emC_LUC[LUC_Num].SCADA.Out.BmsUdcAct	:=	emC_LUC[LUC_Num].BattPLC.CtrlLo.Out.Batt_Sys.BattSysMeasure.UdcAct		;
emC_LUC[LUC_Num].SCADA.Out.BmsIdcAct	:=	emC_LUC[LUC_Num].BattPLC.CtrlLo.Out.Batt_Sys.BattSysMeasure.IdcAct		;
emC_LUC[LUC_Num].SCADA.Out.BmsNomPAct	:=	emC_LUC[LUC_Num].BattPLC.CtrlLo.Out.Batt_Sys.BattSysMeasure.NomPAct		;
emC_LUC[LUC_Num].SCADA.Out.BmsNomEAct	:=	emC_LUC[LUC_Num].BattPLC.CtrlLo.Out.Batt_Sys.BattSysMeasure.NomEAct		;
emC_LUC[LUC_Num].SCADA.Out.BatPNomMaxAct	:=	emC_LUC[LUC_Num].BattPLC.CtrlLo.Out.Batt_Sys.BattSysMeasure.BatPNomMaxAct		;
emC_LUC[LUC_Num].SCADA.Out.BatPNomMinAct	:=	emC_LUC[LUC_Num].BattPLC.CtrlLo.Out.Batt_Sys.BattSysMeasure.BatPNomMinAct		;
emC_LUC[LUC_Num].SCADA.Out.BmsPAct	:=	emC_LUC[LUC_Num].BattPLC.CtrlLo.Out.Batt_Sys.BattSysMeasure.PAct		;
emC_LUC[LUC_Num].SCADA.Out.BmsEAct	:=	emC_LUC[LUC_Num].BattPLC.CtrlLo.Out.Batt_Sys.BattSysMeasure.EAct		;
emC_LUC[LUC_Num].SCADA.Out.BmsSocPctAct	:=	emC_LUC[LUC_Num].BattPLC.CtrlLo.Out.Batt_Sys.BattSysMeasure.SocPctAct		;
emC_LUC[LUC_Num].SCADA.Out.BmsSohAct	:=	emC_LUC[LUC_Num].BattPLC.CtrlLo.Out.Batt_Sys.BattSysMeasure.SohAct		;
emC_LUC[LUC_Num].SCADA.Out.BmsTempMaxAct	:=	emC_LUC[LUC_Num].BattPLC.CtrlLo.Out.Batt_Sys.BattSysMeasure.TempMaxAct		;
emC_LUC[LUC_Num].SCADA.Out.BmsTempMinAct	:=	emC_LUC[LUC_Num].BattPLC.CtrlLo.Out.Batt_Sys.BattSysMeasure.TempMinAct		;
emC_LUC[LUC_Num].SCADA.Out.BmsSyncUSet	:=	emC_LUC[LUC_Num].BattPLC.CtrlLo.Out.Batt_Sys.BattSysMeasure.SyncUSet		;
emC_LUC[LUC_Num].SCADA.Out.BmsHeartBeat	:=	emC_LUC[LUC_Num].BattPLC.CtrlLo.Out.Batt_Sys.BMS_DATA.HeartBeat		;
emC_LUC[LUC_Num].SCADA.Out.BmsVersion	:=	UINT_TO_REAL(emC_LUC[LUC_Num].BattPLC.CtrlLo.Out.Batt_Sys.BMS_DATA.Version	)	;
emC_LUC[LUC_Num].SCADA.Out.BmsRacksNServiceCnt	:=	USINT_TO_REAL(emC_LUC[LUC_Num].BattPLC.CtrlLo.Out.Batt_Sys.BMS_DATA.RacksNServiceCnt)		;
emC_LUC[LUC_Num].SCADA.Out.BmsTotalRackCnt	:=	USINT_TO_REAL(emC_LUC[LUC_Num].BattPLC.CtrlLo.Out.Batt_Sys.BMS_DATA.TotalRackCnt)		;
emC_LUC[LUC_Num].SCADA.Out.BmsPartMinRackCnt	:=	USINT_TO_REAL(emC_LUC[LUC_Num].BattPLC.CtrlLo.Out.Batt_Sys.BMS_DATA.PartMinRackCnt)		;
								
								
								
								
								
emC_LUC[LUC_Num].SCADA.Out.PSStateWord	:=	INT_TO_REAL(emC_LUC[LUC_Num].emPs.PS.PSStateWord)	;
emC_LUC[LUC_Num].SCADA.Out.GCABBStateWord	:=	INT_TO_REAL(emC_LUC[LUC_Num].emPs.PS.ABBStateWord)	;
emC_LUC[LUC_Num].SCADA.Out.GCPAct	:=	emC_LUC[LUC_Num].emPs.PS.GCPAct	;
emC_LUC[LUC_Num].SCADA.Out.GCFAct	:=	emC_LUC[LUC_Num].emPs.PS.GCFAct	;
emC_LUC[LUC_Num].SCADA.Out.GCSNomAct	:=	emC_LUC[LUC_Num].emPs.PS.GCSNomAct	;
emC_LUC[LUC_Num].SCADA.Out.GCQAct	:=	emC_LUC[LUC_Num].emPs.PS.GCQAct	;
emC_LUC[LUC_Num].SCADA.Out.GCPF	:=	emC_LUC[LUC_Num].emPs.PS.GCPF	;
emC_LUC[LUC_Num].SCADA.Out.GCEAct	:=	emC_LUC[LUC_Num].emPs.PS.GCEAct	;
emC_LUC[LUC_Num].SCADA.Out.GCTempAct	:=	emC_LUC[LUC_Num].emPs.PS.TempAct	;
emC_LUC[LUC_Num].SCADA.Out.GCIGBTTempaAct	:=	emC_LUC[LUC_Num].emPs.PS.IGBTTempaAct	;
emC_LUC[LUC_Num].SCADA.Out.GCTrafoTempAct	:=	emC_LUC[LUC_Num].emPs.PS.TrafoTempAct	;
emC_LUC[LUC_Num].SCADA.Out.GCOTTempAct	:=	emC_LUC[LUC_Num].emPs.PS.OTTempAct	;
emC_LUC[LUC_Num].SCADA.Out.GCUAct12	:=	emC_LUC[LUC_Num].emPs.PS.GCUAct12	;
emC_LUC[LUC_Num].SCADA.Out.GCUAct23	:=	emC_LUC[LUC_Num].emPs.PS.GCUAct23	;
emC_LUC[LUC_Num].SCADA.Out.GCUAct13	:=	emC_LUC[LUC_Num].emPs.PS.GCUAct13	;
emC_LUC[LUC_Num].SCADA.Out.GCUAct1N	:=	emC_LUC[LUC_Num].emPs.PS.GCUAct1N	;
emC_LUC[LUC_Num].SCADA.Out.GCUAct2N	:=	emC_LUC[LUC_Num].emPs.PS.GCUAct2N	;
emC_LUC[LUC_Num].SCADA.Out.GCUAct3N	:=	emC_LUC[LUC_Num].emPs.PS.GCUAct3N	;
emC_LUC[LUC_Num].SCADA.Out.GCUAct	:=	emC_LUC[LUC_Num].emPs.PS.GCUAct	;
emC_LUC[LUC_Num].SCADA.Out.GCABBErrorID	:=	emC_LUC[LUC_Num].emPs.PS.GCABBErrorID	;
emC_LUC[LUC_Num].SCADA.Out.GCSysFltCode	:=	UINT_TO_REAL(emC_LUC[LUC_Num].emPs.PS.GCSysFltCode)	;
emC_LUC[LUC_Num].SCADA.Out.I1Act	:=	emC_LUC[LUC_Num].emPs.PS.GCAPhA	;
emC_LUC[LUC_Num].SCADA.Out.I2Act	:=	emC_LUC[LUC_Num].emPs.PS.GCAPhB	;
emC_LUC[LUC_Num].SCADA.Out.I3Act	:=	emC_LUC[LUC_Num].emPs.PS.GCAPhC	;
								
								
								
S_MFI_MNG_16	(MFI_Value:=	emC_LUC[LUC_Num].SCADA.Out.GcSPNomAct	,TimeTag:=Timestamp,IV:=FALSE,CycTrigPa:=FALSE,DeadBTransmitPa:=REAL#0.0,TransmitModePa:= INT#1);	GcSPNomAct_Q	:=	S_MFI_MNG_16.Analog_Output_Q	;
S_MFI_MNG_17	(MFI_Value:=	emC_LUC[LUC_Num].SCADA.Out.GcINomAct	,TimeTag:=Timestamp,IV:=FALSE,CycTrigPa:=FALSE,DeadBTransmitPa:=REAL#0.0,TransmitModePa:= INT#1);	GcINomAct_Q	:=	S_MFI_MNG_17.Analog_Output_Q	;
S_MFI_MNG_18	(MFI_Value:=	emC_LUC[LUC_Num].SCADA.Out.GcUNomAct	,TimeTag:=Timestamp,IV:=FALSE,CycTrigPa:=FALSE,DeadBTransmitPa:=REAL#0.0,TransmitModePa:= INT#1);	GcUNomAct_Q	:=	S_MFI_MNG_18.Analog_Output_Q	;
S_MFI_MNG_19	(MFI_Value:=	emC_LUC[LUC_Num].SCADA.Out.GcFNomAct	,TimeTag:=Timestamp,IV:=FALSE,CycTrigPa:=FALSE,DeadBTransmitPa:=REAL#0.0,TransmitModePa:= INT#1);	GcFNomAct_Q	:=	S_MFI_MNG_19.Analog_Output_Q	;
S_MFI_MNG_20	(MFI_Value:=	emC_LUC[LUC_Num].SCADA.Out.GcModUNomAct	,TimeTag:=Timestamp,IV:=FALSE,CycTrigPa:=FALSE,DeadBTransmitPa:=REAL#0.0,TransmitModePa:= INT#1);	GcModUNomAct_Q	:=	S_MFI_MNG_20.Analog_Output_Q	;
								
S_MFI_MNG_21	(MFI_Value:=	emC_LUC[LUC_Num].SCADA.Out.BmsUdcAct	,TimeTag:=Timestamp,IV:=FALSE,CycTrigPa:=FALSE,DeadBTransmitPa:=REAL#0.0,TransmitModePa:= INT#1);	BmsUdcAct_Q	:=	S_MFI_MNG_21.Analog_Output_Q	;
S_MFI_MNG_22	(MFI_Value:=	emC_LUC[LUC_Num].SCADA.Out.BmsIdcAct	,TimeTag:=Timestamp,IV:=FALSE,CycTrigPa:=FALSE,DeadBTransmitPa:=REAL#0.0,TransmitModePa:= INT#1);	BmsIdcAct_Q	:=	S_MFI_MNG_22.Analog_Output_Q	;
S_MFI_MNG_23	(MFI_Value:=	emC_LUC[LUC_Num].SCADA.Out.BmsNomPAct	,TimeTag:=Timestamp,IV:=FALSE,CycTrigPa:=FALSE,DeadBTransmitPa:=REAL#0.0,TransmitModePa:= INT#1);	BmsNomPAct_Q	:=	S_MFI_MNG_23.Analog_Output_Q	;
S_MFI_MNG_24	(MFI_Value:=	emC_LUC[LUC_Num].SCADA.Out.BmsNomEAct	,TimeTag:=Timestamp,IV:=FALSE,CycTrigPa:=FALSE,DeadBTransmitPa:=REAL#0.0,TransmitModePa:= INT#1);	BmsNomEAct_Q	:=	S_MFI_MNG_24.Analog_Output_Q	;
S_MFI_MNG_25	(MFI_Value:=	emC_LUC[LUC_Num].SCADA.Out.BatPNomMaxAct	,TimeTag:=Timestamp,IV:=FALSE,CycTrigPa:=FALSE,DeadBTransmitPa:=REAL#0.0,TransmitModePa:= INT#1);	BmsBatPNomMaxAct_Q	:=	S_MFI_MNG_25.Analog_Output_Q	;
S_MFI_MNG_26	(MFI_Value:=	emC_LUC[LUC_Num].SCADA.Out.BatPNomMinAct	,TimeTag:=Timestamp,IV:=FALSE,CycTrigPa:=FALSE,DeadBTransmitPa:=REAL#0.0,TransmitModePa:= INT#1);	BmsBatPNomMinAct_Q	:=	S_MFI_MNG_26.Analog_Output_Q	;
S_MFI_MNG_27	(MFI_Value:=	emC_LUC[LUC_Num].SCADA.Out.BmsPAct	,TimeTag:=Timestamp,IV:=FALSE,CycTrigPa:=FALSE,DeadBTransmitPa:=REAL#0.0,TransmitModePa:= INT#1);	BmsPAct_Q	:=	S_MFI_MNG_27.Analog_Output_Q	;
S_MFI_MNG_28	(MFI_Value:=	emC_LUC[LUC_Num].SCADA.Out.BmsEAct	,TimeTag:=Timestamp,IV:=FALSE,CycTrigPa:=FALSE,DeadBTransmitPa:=REAL#0.0,TransmitModePa:= INT#1);	BmsEAct_Q	:=	S_MFI_MNG_28.Analog_Output_Q	;
S_MFI_MNG_29	(MFI_Value:=	emC_LUC[LUC_Num].SCADA.Out.BmsSocPctAct	,TimeTag:=Timestamp,IV:=FALSE,CycTrigPa:=FALSE,DeadBTransmitPa:=REAL#0.0,TransmitModePa:= INT#1);	BatSocAct_Q	:=	S_MFI_MNG_29.Analog_Output_Q	;
S_MFI_MNG_30	(MFI_Value:=	emC_LUC[LUC_Num].SCADA.Out.BmsSohAct	,TimeTag:=Timestamp,IV:=FALSE,CycTrigPa:=FALSE,DeadBTransmitPa:=REAL#0.0,TransmitModePa:= INT#1);	BmsSohAct_Q	:=	S_MFI_MNG_30.Analog_Output_Q	;
S_MFI_MNG_31	(MFI_Value:=	emC_LUC[LUC_Num].SCADA.Out.BmsTempMaxAct	,TimeTag:=Timestamp,IV:=FALSE,CycTrigPa:=FALSE,DeadBTransmitPa:=REAL#0.0,TransmitModePa:= INT#1);	BmsTempMaxAct_Q	:=	S_MFI_MNG_31.Analog_Output_Q	;
S_MFI_MNG_32	(MFI_Value:=	emC_LUC[LUC_Num].SCADA.Out.BmsTempMinAct	,TimeTag:=Timestamp,IV:=FALSE,CycTrigPa:=FALSE,DeadBTransmitPa:=REAL#0.0,TransmitModePa:= INT#1);	BmsTempMinAct_Q	:=	S_MFI_MNG_32.Analog_Output_Q	;
S_MFI_MNG_33	(MFI_Value:=	emC_LUC[LUC_Num].SCADA.Out.BmsSyncUSet	,TimeTag:=Timestamp,IV:=FALSE,CycTrigPa:=FALSE,DeadBTransmitPa:=REAL#0.0,TransmitModePa:= INT#1);	BmsSyncUSet_Q	:=	S_MFI_MNG_33.Analog_Output_Q	;
S_MFI_MNG_34	(MFI_Value:=	emC_LUC[LUC_Num].SCADA.Out.BmsHeartBeat	,TimeTag:=Timestamp,IV:=FALSE,CycTrigPa:=FALSE,DeadBTransmitPa:=REAL#0.0,TransmitModePa:= INT#1);	BmsHeartBeat_Q	:=	S_MFI_MNG_34.Analog_Output_Q	;							
S_MFI_MNG_37	(MFI_Value:=	emC_LUC[LUC_Num].SCADA.Out.BmsVersion	,TimeTag:=Timestamp,IV:=FALSE,CycTrigPa:=FALSE,DeadBTransmitPa:=REAL#0.0,TransmitModePa:= INT#1);	BmsVersion_Q	:=	S_MFI_MNG_37.Analog_Output_Q	;
S_MFI_MNG_38	(MFI_Value:=	emC_LUC[LUC_Num].SCADA.Out.BmsRacksNServiceCnt	,TimeTag:=Timestamp,IV:=FALSE,CycTrigPa:=FALSE,DeadBTransmitPa:=REAL#0.0,TransmitModePa:= INT#1);	BmsRacksNServiceCnt_Q	:=	S_MFI_MNG_38.Analog_Output_Q	;
S_MFI_MNG_39	(MFI_Value:=	emC_LUC[LUC_Num].SCADA.Out.BmsTotalRackCnt	,TimeTag:=Timestamp,IV:=FALSE,CycTrigPa:=FALSE,DeadBTransmitPa:=REAL#0.0,TransmitModePa:= INT#1);	BmsTotalRackCnt_Q	:=	S_MFI_MNG_39.Analog_Output_Q	;
S_MFI_MNG_40	(MFI_Value:=	emC_LUC[LUC_Num].SCADA.Out.BmsPartMinRackCnt	,TimeTag:=Timestamp,IV:=FALSE,CycTrigPa:=FALSE,DeadBTransmitPa:=REAL#0.0,TransmitModePa:= INT#1);	BmsPartMinRackCnt_Q	:=	S_MFI_MNG_40.Analog_Output_Q	;
								
								
								
							
S_MFI_MNG_41	(MFI_Value:=	emC_LUC[LUC_Num].SCADA.Out.PSStateWord	,TimeTag:=Timestamp,IV:=FALSE,CycTrigPa:=FALSE,DeadBTransmitPa:=REAL#0.0,TransmitModePa:= INT#1);	PSStateWord_Q	:=	S_MFI_MNG_41.Analog_Output_Q	;
S_MFI_MNG_42	(MFI_Value:=	emC_LUC[LUC_Num].SCADA.Out.GCABBStateWord	,TimeTag:=Timestamp,IV:=FALSE,CycTrigPa:=FALSE,DeadBTransmitPa:=REAL#0.0,TransmitModePa:= INT#1);	ABBStateWord_Q	:=	S_MFI_MNG_42.Analog_Output_Q	;
S_MFI_MNG_43	(MFI_Value:=	emC_LUC[LUC_Num].SCADA.Out.GCPAct	,TimeTag:=Timestamp,IV:=FALSE,CycTrigPa:=FALSE,DeadBTransmitPa:=REAL#0.0,TransmitModePa:= INT#1);	GCPAct_Q	:=	S_MFI_MNG_43.Analog_Output_Q	;
S_MFI_MNG_44	(MFI_Value:=	emC_LUC[LUC_Num].SCADA.Out.GCFAct	,TimeTag:=Timestamp,IV:=FALSE,CycTrigPa:=FALSE,DeadBTransmitPa:=REAL#0.0,TransmitModePa:= INT#1);	GCFAct_Q	:=	S_MFI_MNG_44.Analog_Output_Q	;
S_MFI_MNG_45	(MFI_Value:=	emC_LUC[LUC_Num].SCADA.Out.GCSNomAct	,TimeTag:=Timestamp,IV:=FALSE,CycTrigPa:=FALSE,DeadBTransmitPa:=REAL#0.0,TransmitModePa:= INT#1);	GCSNomAct_Q	:=	S_MFI_MNG_45.Analog_Output_Q	;
S_MFI_MNG_46	(MFI_Value:=	emC_LUC[LUC_Num].SCADA.Out.GCQAct	,TimeTag:=Timestamp,IV:=FALSE,CycTrigPa:=FALSE,DeadBTransmitPa:=REAL#0.0,TransmitModePa:= INT#1);	GCQAct_Q	:=	S_MFI_MNG_46.Analog_Output_Q	;
S_MFI_MNG_47	(MFI_Value:=	emC_LUC[LUC_Num].SCADA.Out.GCPF	,TimeTag:=Timestamp,IV:=FALSE,CycTrigPa:=FALSE,DeadBTransmitPa:=REAL#0.0,TransmitModePa:= INT#1);	GCPF_Q	:=	S_MFI_MNG_47.Analog_Output_Q	;
S_MFI_MNG_48	(MFI_Value:=	emC_LUC[LUC_Num].SCADA.Out.GCEAct	,TimeTag:=Timestamp,IV:=FALSE,CycTrigPa:=FALSE,DeadBTransmitPa:=REAL#0.0,TransmitModePa:= INT#1);	GCEAct_Q	:=	S_MFI_MNG_48.Analog_Output_Q	;
S_MFI_MNG_49	(MFI_Value:=	emC_LUC[LUC_Num].SCADA.Out.GCTempAct	,TimeTag:=Timestamp,IV:=FALSE,CycTrigPa:=FALSE,DeadBTransmitPa:=REAL#0.0,TransmitModePa:= INT#1);	TempAct_Q	:=	S_MFI_MNG_49.Analog_Output_Q	;
S_MFI_MNG_50	(MFI_Value:=	emC_LUC[LUC_Num].SCADA.Out.GCIGBTTempaAct	,TimeTag:=Timestamp,IV:=FALSE,CycTrigPa:=FALSE,DeadBTransmitPa:=REAL#0.0,TransmitModePa:= INT#1);	IGBTTempaAct_Q	:=	S_MFI_MNG_50.Analog_Output_Q	;
S_MFI_MNG_51	(MFI_Value:=	emC_LUC[LUC_Num].SCADA.Out.GCTrafoTempAct	,TimeTag:=Timestamp,IV:=FALSE,CycTrigPa:=FALSE,DeadBTransmitPa:=REAL#0.0,TransmitModePa:= INT#1);	TrafoTempAct_Q	:=	S_MFI_MNG_51.Analog_Output_Q	;
S_MFI_MNG_52	(MFI_Value:=	emC_LUC[LUC_Num].SCADA.Out.GCOTTempAct	,TimeTag:=Timestamp,IV:=FALSE,CycTrigPa:=FALSE,DeadBTransmitPa:=REAL#0.0,TransmitModePa:= INT#1);	OTTempAct_Q	:=	S_MFI_MNG_52.Analog_Output_Q	;
S_MFI_MNG_53	(MFI_Value:=	emC_LUC[LUC_Num].SCADA.Out.GCUAct12	,TimeTag:=Timestamp,IV:=FALSE,CycTrigPa:=FALSE,DeadBTransmitPa:=REAL#0.0,TransmitModePa:= INT#1);	GCUAct12_Q	:=	S_MFI_MNG_53.Analog_Output_Q	;
S_MFI_MNG_54	(MFI_Value:=	emC_LUC[LUC_Num].SCADA.Out.GCUAct23	,TimeTag:=Timestamp,IV:=FALSE,CycTrigPa:=FALSE,DeadBTransmitPa:=REAL#0.0,TransmitModePa:= INT#1);	GCUAct23_Q	:=	S_MFI_MNG_54.Analog_Output_Q	;
S_MFI_MNG_55	(MFI_Value:=	emC_LUC[LUC_Num].SCADA.Out.GCUAct13	,TimeTag:=Timestamp,IV:=FALSE,CycTrigPa:=FALSE,DeadBTransmitPa:=REAL#0.0,TransmitModePa:= INT#1);	GCUAct13_Q	:=	S_MFI_MNG_55.Analog_Output_Q	;
S_MFI_MNG_56	(MFI_Value:=	emC_LUC[LUC_Num].SCADA.Out.GCUAct1N	,TimeTag:=Timestamp,IV:=FALSE,CycTrigPa:=FALSE,DeadBTransmitPa:=REAL#0.0,TransmitModePa:= INT#1);	GCUAct1N_Q	:=	S_MFI_MNG_56.Analog_Output_Q	;
S_MFI_MNG_57	(MFI_Value:=	emC_LUC[LUC_Num].SCADA.Out.GCUAct2N	,TimeTag:=Timestamp,IV:=FALSE,CycTrigPa:=FALSE,DeadBTransmitPa:=REAL#0.0,TransmitModePa:= INT#1);	GCUAct2N_Q	:=	S_MFI_MNG_57.Analog_Output_Q	;
S_MFI_MNG_58	(MFI_Value:=	emC_LUC[LUC_Num].SCADA.Out.GCUAct3N	,TimeTag:=Timestamp,IV:=FALSE,CycTrigPa:=FALSE,DeadBTransmitPa:=REAL#0.0,TransmitModePa:= INT#1);	GCUAct3N_Q	:=	S_MFI_MNG_58.Analog_Output_Q	;
S_MFI_MNG_59	(MFI_Value:=	emC_LUC[LUC_Num].SCADA.Out.GCUAct	,TimeTag:=Timestamp,IV:=FALSE,CycTrigPa:=FALSE,DeadBTransmitPa:=REAL#0.0,TransmitModePa:= INT#1);	GCUAct_Q	:=	S_MFI_MNG_59.Analog_Output_Q	;
S_MFI_MNG_60	(MFI_Value:=	emC_LUC[LUC_Num].SCADA.Out.GCABBErrorID	,TimeTag:=Timestamp,IV:=FALSE,CycTrigPa:=FALSE,DeadBTransmitPa:=REAL#0.0,TransmitModePa:= INT#1);	GCABBErrorID_Q	:=	S_MFI_MNG_60.Analog_Output_Q	;
S_MFI_MNG_61	(MFI_Value:=	emC_LUC[LUC_Num].SCADA.Out.GCSysFltCode	,TimeTag:=Timestamp,IV:=FALSE,CycTrigPa:=FALSE,DeadBTransmitPa:=REAL#0.0,TransmitModePa:= INT#1);	GCSysFltCode_Q	:=	S_MFI_MNG_61.Analog_Output_Q	;
								
S_MFI_MNG_62	(MFI_Value:=	emC_LUC[LUC_Num].SCADA.Out.I1Act	,TimeTag:=Timestamp,IV:=FALSE,CycTrigPa:=FALSE,DeadBTransmitPa:=REAL#0.0,TransmitModePa:= INT#1);	GCI1_Q	:=	S_MFI_MNG_62.Analog_Output_Q	;
S_MFI_MNG_63	(MFI_Value:=	emC_LUC[LUC_Num].SCADA.Out.I2Act	,TimeTag:=Timestamp,IV:=FALSE,CycTrigPa:=FALSE,DeadBTransmitPa:=REAL#0.0,TransmitModePa:= INT#1);	GCI2_Q	:=	S_MFI_MNG_63.Analog_Output_Q	;
S_MFI_MNG_64	(MFI_Value:=	emC_LUC[LUC_Num].SCADA.Out.I3Act	,TimeTag:=Timestamp,IV:=FALSE,CycTrigPa:=FALSE,DeadBTransmitPa:=REAL#0.0,TransmitModePa:= INT#1);	GCI3_Q	:=	S_MFI_MNG_64.Analog_Output_Q	;
S_MFI_MNG_65	(MFI_Value:=	emC_LUC[LUC_Num].SCADA.Out.IAvgAct	,TimeTag:=Timestamp,IV:=FALSE,CycTrigPa:=FALSE,DeadBTransmitPa:=REAL#0.0,TransmitModePa:= INT#1);	GCIAvgAct_Q	:=	S_MFI_MNG_64.Analog_Output_Q	;
								
								
								
								
S_SPI_MNG_301	(Digital_Feedback_Value:=	emC_LUC[LUC_Num].SCADA.Out.Rk[1].OnlineSt	,TimeTag:=Timestamp,IV:=FALSE);	Rk1OnlineSt_Q	:=	S_SPI_MNG_301.Digital_Feedback_Q	;
S_SPI_MNG_302	(Digital_Feedback_Value:=	emC_LUC[LUC_Num].SCADA.Out.Rk[1].FaultSt	,TimeTag:=Timestamp,IV:=FALSE);	Rk1FaultSt_Q	:=	S_SPI_MNG_302.Digital_Feedback_Q	;
S_MFI_MNG_303	(MFI_Value:=	emC_LUC[LUC_Num].SCADA.Out.Rk[1].SoCAct	,TimeTag:=Timestamp,IV:=FALSE,CycTrigPa:=FALSE,DeadBTransmitPa:=REAL#0.0,TransmitModePa:= INT#1);	Rk1SoCAct_Q	:=	S_MFI_MNG_303.Analog_Output_Q	;
S_MFI_MNG_304	(MFI_Value:=	emC_LUC[LUC_Num].SCADA.Out.Rk[1].SoHAct	,TimeTag:=Timestamp,IV:=FALSE,CycTrigPa:=FALSE,DeadBTransmitPa:=REAL#0.0,TransmitModePa:= INT#1);	Rk1SoHAct_Q	:=	S_MFI_MNG_304.Analog_Output_Q	;
S_MFI_MNG_305	(MFI_Value:=	emC_LUC[LUC_Num].SCADA.Out.Rk[1].UAct	,TimeTag:=Timestamp,IV:=FALSE,CycTrigPa:=FALSE,DeadBTransmitPa:=REAL#0.0,TransmitModePa:= INT#1);	Rk1UAct_Q	:=	S_MFI_MNG_305.Analog_Output_Q	;
S_MFI_MNG_306	(MFI_Value:=	emC_LUC[LUC_Num].SCADA.Out.Rk[1].IAct	,TimeTag:=Timestamp,IV:=FALSE,CycTrigPa:=FALSE,DeadBTransmitPa:=REAL#0.0,TransmitModePa:= INT#1);	Rk1IAct_Q	:=	S_MFI_MNG_306.Analog_Output_Q	;
S_MFI_MNG_307	(MFI_Value:=	emC_LUC[LUC_Num].SCADA.Out.Rk[1].TempAct	,TimeTag:=Timestamp,IV:=FALSE,CycTrigPa:=FALSE,DeadBTransmitPa:=REAL#0.0,TransmitModePa:= INT#1);	Rk1TempAct_Q	:=	S_MFI_MNG_307.Analog_Output_Q	;
S_SPI_MNG_308	(Digital_Feedback_Value:=	emC_LUC[LUC_Num].SCADA.Out.Rk[2].OnlineSt	,TimeTag:=Timestamp,IV:=FALSE);	Rk2OnlineSt_Q	:=	S_SPI_MNG_308.Digital_Feedback_Q	;
S_SPI_MNG_309	(Digital_Feedback_Value:=	emC_LUC[LUC_Num].SCADA.Out.Rk[2].FaultSt	,TimeTag:=Timestamp,IV:=FALSE);	Rk2FaultSt_Q	:=	S_SPI_MNG_309.Digital_Feedback_Q	;
S_MFI_MNG_310	(MFI_Value:=	emC_LUC[LUC_Num].SCADA.Out.Rk[2].SoCAct	,TimeTag:=Timestamp,IV:=FALSE,CycTrigPa:=FALSE,DeadBTransmitPa:=REAL#0.0,TransmitModePa:= INT#1);	Rk2SoCAct_Q	:=	S_MFI_MNG_310.Analog_Output_Q	;
S_MFI_MNG_311	(MFI_Value:=	emC_LUC[LUC_Num].SCADA.Out.Rk[2].SoHAct	,TimeTag:=Timestamp,IV:=FALSE,CycTrigPa:=FALSE,DeadBTransmitPa:=REAL#0.0,TransmitModePa:= INT#1);	Rk2SoHAct_Q	:=	S_MFI_MNG_311.Analog_Output_Q	;
S_MFI_MNG_312	(MFI_Value:=	emC_LUC[LUC_Num].SCADA.Out.Rk[2].UAct	,TimeTag:=Timestamp,IV:=FALSE,CycTrigPa:=FALSE,DeadBTransmitPa:=REAL#0.0,TransmitModePa:= INT#1);	Rk2UAct_Q	:=	S_MFI_MNG_312.Analog_Output_Q	;
S_MFI_MNG_313	(MFI_Value:=	emC_LUC[LUC_Num].SCADA.Out.Rk[2].IAct	,TimeTag:=Timestamp,IV:=FALSE,CycTrigPa:=FALSE,DeadBTransmitPa:=REAL#0.0,TransmitModePa:= INT#1);	Rk2IAct_Q	:=	S_MFI_MNG_313.Analog_Output_Q	;
S_MFI_MNG_314	(MFI_Value:=	emC_LUC[LUC_Num].SCADA.Out.Rk[2].TempAct	,TimeTag:=Timestamp,IV:=FALSE,CycTrigPa:=FALSE,DeadBTransmitPa:=REAL#0.0,TransmitModePa:= INT#1);	Rk2TempAct_Q	:=	S_MFI_MNG_314.Analog_Output_Q	;
S_SPI_MNG_315	(Digital_Feedback_Value:=	emC_LUC[LUC_Num].SCADA.Out.Rk[3].OnlineSt	,TimeTag:=Timestamp,IV:=FALSE);	Rk3OnlineSt_Q	:=	S_SPI_MNG_315.Digital_Feedback_Q	;
S_SPI_MNG_316	(Digital_Feedback_Value:=	emC_LUC[LUC_Num].SCADA.Out.Rk[3].FaultSt	,TimeTag:=Timestamp,IV:=FALSE);	Rk3FaultSt_Q	:=	S_SPI_MNG_316.Digital_Feedback_Q	;
S_MFI_MNG_317	(MFI_Value:=	emC_LUC[LUC_Num].SCADA.Out.Rk[3].SoCAct	,TimeTag:=Timestamp,IV:=FALSE,CycTrigPa:=FALSE,DeadBTransmitPa:=REAL#0.0,TransmitModePa:= INT#1);	Rk3SoCAct_Q	:=	S_MFI_MNG_317.Analog_Output_Q	;
S_MFI_MNG_318	(MFI_Value:=	emC_LUC[LUC_Num].SCADA.Out.Rk[3].SoHAct	,TimeTag:=Timestamp,IV:=FALSE,CycTrigPa:=FALSE,DeadBTransmitPa:=REAL#0.0,TransmitModePa:= INT#1);	Rk3SoHAct_Q	:=	S_MFI_MNG_318.Analog_Output_Q	;
S_MFI_MNG_319	(MFI_Value:=	emC_LUC[LUC_Num].SCADA.Out.Rk[3].UAct	,TimeTag:=Timestamp,IV:=FALSE,CycTrigPa:=FALSE,DeadBTransmitPa:=REAL#0.0,TransmitModePa:= INT#1);	Rk3UAct_Q	:=	S_MFI_MNG_319.Analog_Output_Q	;
S_MFI_MNG_320	(MFI_Value:=	emC_LUC[LUC_Num].SCADA.Out.Rk[3].IAct	,TimeTag:=Timestamp,IV:=FALSE,CycTrigPa:=FALSE,DeadBTransmitPa:=REAL#0.0,TransmitModePa:= INT#1);	Rk3IAct_Q	:=	S_MFI_MNG_320.Analog_Output_Q	;
S_MFI_MNG_321	(MFI_Value:=	emC_LUC[LUC_Num].SCADA.Out.Rk[3].TempAct	,TimeTag:=Timestamp,IV:=FALSE,CycTrigPa:=FALSE,DeadBTransmitPa:=REAL#0.0,TransmitModePa:= INT#1);	Rk3TempAct_Q	:=	S_MFI_MNG_321.Analog_Output_Q	;
S_SPI_MNG_322	(Digital_Feedback_Value:=	emC_LUC[LUC_Num].SCADA.Out.Rk[4].OnlineSt	,TimeTag:=Timestamp,IV:=FALSE);	Rk4OnlineSt_Q	:=	S_SPI_MNG_322.Digital_Feedback_Q	;
S_SPI_MNG_323	(Digital_Feedback_Value:=	emC_LUC[LUC_Num].SCADA.Out.Rk[4].FaultSt	,TimeTag:=Timestamp,IV:=FALSE);	Rk4FaultSt_Q	:=	S_SPI_MNG_323.Digital_Feedback_Q	;
S_MFI_MNG_324	(MFI_Value:=	emC_LUC[LUC_Num].SCADA.Out.Rk[4].SoCAct	,TimeTag:=Timestamp,IV:=FALSE,CycTrigPa:=FALSE,DeadBTransmitPa:=REAL#0.0,TransmitModePa:= INT#1);	Rk4SoCAct_Q	:=	S_MFI_MNG_324.Analog_Output_Q	;
S_MFI_MNG_325	(MFI_Value:=	emC_LUC[LUC_Num].SCADA.Out.Rk[4].SoHAct	,TimeTag:=Timestamp,IV:=FALSE,CycTrigPa:=FALSE,DeadBTransmitPa:=REAL#0.0,TransmitModePa:= INT#1);	Rk4SoHAct_Q	:=	S_MFI_MNG_325.Analog_Output_Q	;
S_MFI_MNG_326	(MFI_Value:=	emC_LUC[LUC_Num].SCADA.Out.Rk[4].UAct	,TimeTag:=Timestamp,IV:=FALSE,CycTrigPa:=FALSE,DeadBTransmitPa:=REAL#0.0,TransmitModePa:= INT#1);	Rk4UAct_Q	:=	S_MFI_MNG_326.Analog_Output_Q	;
S_MFI_MNG_327	(MFI_Value:=	emC_LUC[LUC_Num].SCADA.Out.Rk[4].IAct	,TimeTag:=Timestamp,IV:=FALSE,CycTrigPa:=FALSE,DeadBTransmitPa:=REAL#0.0,TransmitModePa:= INT#1);	Rk4IAct_Q	:=	S_MFI_MNG_327.Analog_Output_Q	;
S_MFI_MNG_328	(MFI_Value:=	emC_LUC[LUC_Num].SCADA.Out.Rk[4].TempAct	,TimeTag:=Timestamp,IV:=FALSE,CycTrigPa:=FALSE,DeadBTransmitPa:=REAL#0.0,TransmitModePa:= INT#1);	Rk4TempAct_Q	:=	S_MFI_MNG_328.Analog_Output_Q	;
S_SPI_MNG_329	(Digital_Feedback_Value:=	emC_LUC[LUC_Num].SCADA.Out.Rk[5].OnlineSt	,TimeTag:=Timestamp,IV:=FALSE);	Rk5OnlineSt_Q	:=	S_SPI_MNG_329.Digital_Feedback_Q	;
S_SPI_MNG_330	(Digital_Feedback_Value:=	emC_LUC[LUC_Num].SCADA.Out.Rk[5].FaultSt	,TimeTag:=Timestamp,IV:=FALSE);	Rk5FaultSt_Q	:=	S_SPI_MNG_330.Digital_Feedback_Q	;
S_MFI_MNG_331	(MFI_Value:=	emC_LUC[LUC_Num].SCADA.Out.Rk[5].SoCAct	,TimeTag:=Timestamp,IV:=FALSE,CycTrigPa:=FALSE,DeadBTransmitPa:=REAL#0.0,TransmitModePa:= INT#1);	Rk5SoCAct_Q	:=	S_MFI_MNG_331.Analog_Output_Q	;
S_MFI_MNG_332	(MFI_Value:=	emC_LUC[LUC_Num].SCADA.Out.Rk[5].SoHAct	,TimeTag:=Timestamp,IV:=FALSE,CycTrigPa:=FALSE,DeadBTransmitPa:=REAL#0.0,TransmitModePa:= INT#1);	Rk5SoHAct_Q	:=	S_MFI_MNG_332.Analog_Output_Q	;
S_MFI_MNG_333	(MFI_Value:=	emC_LUC[LUC_Num].SCADA.Out.Rk[5].UAct	,TimeTag:=Timestamp,IV:=FALSE,CycTrigPa:=FALSE,DeadBTransmitPa:=REAL#0.0,TransmitModePa:= INT#1);	Rk5UAct_Q	:=	S_MFI_MNG_333.Analog_Output_Q	;
S_MFI_MNG_334	(MFI_Value:=	emC_LUC[LUC_Num].SCADA.Out.Rk[5].IAct	,TimeTag:=Timestamp,IV:=FALSE,CycTrigPa:=FALSE,DeadBTransmitPa:=REAL#0.0,TransmitModePa:= INT#1);	Rk5IAct_Q	:=	S_MFI_MNG_334.Analog_Output_Q	;
S_MFI_MNG_335	(MFI_Value:=	emC_LUC[LUC_Num].SCADA.Out.Rk[5].TempAct	,TimeTag:=Timestamp,IV:=FALSE,CycTrigPa:=FALSE,DeadBTransmitPa:=REAL#0.0,TransmitModePa:= INT#1);	Rk5TempAct_Q	:=	S_MFI_MNG_335.Analog_Output_Q	;
S_SPI_MNG_336	(Digital_Feedback_Value:=	emC_LUC[LUC_Num].SCADA.Out.Rk[6].OnlineSt	,TimeTag:=Timestamp,IV:=FALSE);	Rk6OnlineSt_Q	:=	S_SPI_MNG_336.Digital_Feedback_Q	;
S_SPI_MNG_337	(Digital_Feedback_Value:=	emC_LUC[LUC_Num].SCADA.Out.Rk[6].FaultSt	,TimeTag:=Timestamp,IV:=FALSE);	Rk6FaultSt_Q	:=	S_SPI_MNG_337.Digital_Feedback_Q	;
S_MFI_MNG_338	(MFI_Value:=	emC_LUC[LUC_Num].SCADA.Out.Rk[6].SoCAct	,TimeTag:=Timestamp,IV:=FALSE,CycTrigPa:=FALSE,DeadBTransmitPa:=REAL#0.0,TransmitModePa:= INT#1);	Rk6SoCAct_Q	:=	S_MFI_MNG_338.Analog_Output_Q	;
S_MFI_MNG_339	(MFI_Value:=	emC_LUC[LUC_Num].SCADA.Out.Rk[6].SoHAct	,TimeTag:=Timestamp,IV:=FALSE,CycTrigPa:=FALSE,DeadBTransmitPa:=REAL#0.0,TransmitModePa:= INT#1);	Rk6SoHAct_Q	:=	S_MFI_MNG_339.Analog_Output_Q	;
S_MFI_MNG_340	(MFI_Value:=	emC_LUC[LUC_Num].SCADA.Out.Rk[6].UAct	,TimeTag:=Timestamp,IV:=FALSE,CycTrigPa:=FALSE,DeadBTransmitPa:=REAL#0.0,TransmitModePa:= INT#1);	Rk6UAct_Q	:=	S_MFI_MNG_340.Analog_Output_Q	;
S_MFI_MNG_341	(MFI_Value:=	emC_LUC[LUC_Num].SCADA.Out.Rk[6].IAct	,TimeTag:=Timestamp,IV:=FALSE,CycTrigPa:=FALSE,DeadBTransmitPa:=REAL#0.0,TransmitModePa:= INT#1);	Rk6IAct_Q	:=	S_MFI_MNG_341.Analog_Output_Q	;
S_MFI_MNG_342	(MFI_Value:=	emC_LUC[LUC_Num].SCADA.Out.Rk[6].TempAct	,TimeTag:=Timestamp,IV:=FALSE,CycTrigPa:=FALSE,DeadBTransmitPa:=REAL#0.0,TransmitModePa:= INT#1);	Rk6TempAct_Q	:=	S_MFI_MNG_342.Analog_Output_Q	;
S_SPI_MNG_343	(Digital_Feedback_Value:=	emC_LUC[LUC_Num].SCADA.Out.Rk[7].OnlineSt	,TimeTag:=Timestamp,IV:=FALSE);	Rk7OnlineSt_Q	:=	S_SPI_MNG_343.Digital_Feedback_Q	;
S_SPI_MNG_344	(Digital_Feedback_Value:=	emC_LUC[LUC_Num].SCADA.Out.Rk[7].FaultSt	,TimeTag:=Timestamp,IV:=FALSE);	Rk7FaultSt_Q	:=	S_SPI_MNG_344.Digital_Feedback_Q	;
S_MFI_MNG_345	(MFI_Value:=	emC_LUC[LUC_Num].SCADA.Out.Rk[7].SoCAct	,TimeTag:=Timestamp,IV:=FALSE,CycTrigPa:=FALSE,DeadBTransmitPa:=REAL#0.0,TransmitModePa:= INT#1);	Rk7SoCAct_Q	:=	S_MFI_MNG_345.Analog_Output_Q	;
S_MFI_MNG_346	(MFI_Value:=	emC_LUC[LUC_Num].SCADA.Out.Rk[7].SoHAct	,TimeTag:=Timestamp,IV:=FALSE,CycTrigPa:=FALSE,DeadBTransmitPa:=REAL#0.0,TransmitModePa:= INT#1);	Rk7SoHAct_Q	:=	S_MFI_MNG_346.Analog_Output_Q	;
S_MFI_MNG_347	(MFI_Value:=	emC_LUC[LUC_Num].SCADA.Out.Rk[7].UAct	,TimeTag:=Timestamp,IV:=FALSE,CycTrigPa:=FALSE,DeadBTransmitPa:=REAL#0.0,TransmitModePa:= INT#1);	Rk7UAct_Q	:=	S_MFI_MNG_347.Analog_Output_Q	;
S_MFI_MNG_348	(MFI_Value:=	emC_LUC[LUC_Num].SCADA.Out.Rk[7].IAct	,TimeTag:=Timestamp,IV:=FALSE,CycTrigPa:=FALSE,DeadBTransmitPa:=REAL#0.0,TransmitModePa:= INT#1);	Rk7IAct_Q	:=	S_MFI_MNG_348.Analog_Output_Q	;
S_MFI_MNG_349	(MFI_Value:=	emC_LUC[LUC_Num].SCADA.Out.Rk[7].TempAct	,TimeTag:=Timestamp,IV:=FALSE,CycTrigPa:=FALSE,DeadBTransmitPa:=REAL#0.0,TransmitModePa:= INT#1);	Rk7TempAct_Q	:=	S_MFI_MNG_349.Analog_Output_Q	;
S_SPI_MNG_350	(Digital_Feedback_Value:=	emC_LUC[LUC_Num].SCADA.Out.Rk[8].OnlineSt	,TimeTag:=Timestamp,IV:=FALSE);	Rk8OnlineSt_Q	:=	S_SPI_MNG_350.Digital_Feedback_Q	;
S_SPI_MNG_351	(Digital_Feedback_Value:=	emC_LUC[LUC_Num].SCADA.Out.Rk[8].FaultSt	,TimeTag:=Timestamp,IV:=FALSE);	Rk8FaultSt_Q	:=	S_SPI_MNG_351.Digital_Feedback_Q	;
S_MFI_MNG_352	(MFI_Value:=	emC_LUC[LUC_Num].SCADA.Out.Rk[8].SoCAct	,TimeTag:=Timestamp,IV:=FALSE,CycTrigPa:=FALSE,DeadBTransmitPa:=REAL#0.0,TransmitModePa:= INT#1);	Rk8SoCAct_Q	:=	S_MFI_MNG_352.Analog_Output_Q	;
S_MFI_MNG_353	(MFI_Value:=	emC_LUC[LUC_Num].SCADA.Out.Rk[8].SoHAct	,TimeTag:=Timestamp,IV:=FALSE,CycTrigPa:=FALSE,DeadBTransmitPa:=REAL#0.0,TransmitModePa:= INT#1);	Rk8SoHAct_Q	:=	S_MFI_MNG_353.Analog_Output_Q	;
S_MFI_MNG_354	(MFI_Value:=	emC_LUC[LUC_Num].SCADA.Out.Rk[8].UAct	,TimeTag:=Timestamp,IV:=FALSE,CycTrigPa:=FALSE,DeadBTransmitPa:=REAL#0.0,TransmitModePa:= INT#1);	Rk8UAct_Q	:=	S_MFI_MNG_354.Analog_Output_Q	;
S_MFI_MNG_355	(MFI_Value:=	emC_LUC[LUC_Num].SCADA.Out.Rk[8].IAct	,TimeTag:=Timestamp,IV:=FALSE,CycTrigPa:=FALSE,DeadBTransmitPa:=REAL#0.0,TransmitModePa:= INT#1);	Rk8IAct_Q	:=	S_MFI_MNG_355.Analog_Output_Q	;
S_MFI_MNG_356	(MFI_Value:=	emC_LUC[LUC_Num].SCADA.Out.Rk[8].TempAct	,TimeTag:=Timestamp,IV:=FALSE,CycTrigPa:=FALSE,DeadBTransmitPa:=REAL#0.0,TransmitModePa:= INT#1);	Rk8TempAct_Q	:=	S_MFI_MNG_356.Analog_Output_Q	;
S_SPI_MNG_357	(Digital_Feedback_Value:=	emC_LUC[LUC_Num].SCADA.Out.Rk[9].OnlineSt	,TimeTag:=Timestamp,IV:=FALSE);	Rk9OnlineSt_Q	:=	S_SPI_MNG_357.Digital_Feedback_Q	;
S_SPI_MNG_358	(Digital_Feedback_Value:=	emC_LUC[LUC_Num].SCADA.Out.Rk[9].FaultSt	,TimeTag:=Timestamp,IV:=FALSE);	Rk9FaultSt_Q	:=	S_SPI_MNG_358.Digital_Feedback_Q	;
S_MFI_MNG_359	(MFI_Value:=	emC_LUC[LUC_Num].SCADA.Out.Rk[9].SoCAct	,TimeTag:=Timestamp,IV:=FALSE,CycTrigPa:=FALSE,DeadBTransmitPa:=REAL#0.0,TransmitModePa:= INT#1);	Rk9SoCAct_Q	:=	S_MFI_MNG_359.Analog_Output_Q	;
S_MFI_MNG_360	(MFI_Value:=	emC_LUC[LUC_Num].SCADA.Out.Rk[9].SoHAct	,TimeTag:=Timestamp,IV:=FALSE,CycTrigPa:=FALSE,DeadBTransmitPa:=REAL#0.0,TransmitModePa:= INT#1);	Rk9SoHAct_Q	:=	S_MFI_MNG_360.Analog_Output_Q	;
S_MFI_MNG_361	(MFI_Value:=	emC_LUC[LUC_Num].SCADA.Out.Rk[9].UAct	,TimeTag:=Timestamp,IV:=FALSE,CycTrigPa:=FALSE,DeadBTransmitPa:=REAL#0.0,TransmitModePa:= INT#1);	Rk9UAct_Q	:=	S_MFI_MNG_361.Analog_Output_Q	;
S_MFI_MNG_362	(MFI_Value:=	emC_LUC[LUC_Num].SCADA.Out.Rk[9].IAct	,TimeTag:=Timestamp,IV:=FALSE,CycTrigPa:=FALSE,DeadBTransmitPa:=REAL#0.0,TransmitModePa:= INT#1);	Rk9IAct_Q	:=	S_MFI_MNG_362.Analog_Output_Q	;
S_MFI_MNG_363	(MFI_Value:=	emC_LUC[LUC_Num].SCADA.Out.Rk[9].TempAct	,TimeTag:=Timestamp,IV:=FALSE,CycTrigPa:=FALSE,DeadBTransmitPa:=REAL#0.0,TransmitModePa:= INT#1);	Rk9TempAct_Q	:=	S_MFI_MNG_363.Analog_Output_Q	;
S_SPI_MNG_364	(Digital_Feedback_Value:=	emC_LUC[LUC_Num].SCADA.Out.Rk[10].OnlineSt	,TimeTag:=Timestamp,IV:=FALSE);	Rk10OnlineSt_Q	:=	S_SPI_MNG_364.Digital_Feedback_Q	;
S_SPI_MNG_365	(Digital_Feedback_Value:=	emC_LUC[LUC_Num].SCADA.Out.Rk[10].FaultSt	,TimeTag:=Timestamp,IV:=FALSE);	Rk10FaultSt_Q	:=	S_SPI_MNG_365.Digital_Feedback_Q	;
S_MFI_MNG_366	(MFI_Value:=	emC_LUC[LUC_Num].SCADA.Out.Rk[10].SoCAct	,TimeTag:=Timestamp,IV:=FALSE,CycTrigPa:=FALSE,DeadBTransmitPa:=REAL#0.0,TransmitModePa:= INT#1);	Rk10SoCAct_Q	:=	S_MFI_MNG_366.Analog_Output_Q	;
S_MFI_MNG_367	(MFI_Value:=	emC_LUC[LUC_Num].SCADA.Out.Rk[10].SoHAct	,TimeTag:=Timestamp,IV:=FALSE,CycTrigPa:=FALSE,DeadBTransmitPa:=REAL#0.0,TransmitModePa:= INT#1);	Rk10SoHAct_Q	:=	S_MFI_MNG_367.Analog_Output_Q	;
S_MFI_MNG_368	(MFI_Value:=	emC_LUC[LUC_Num].SCADA.Out.Rk[10].UAct	,TimeTag:=Timestamp,IV:=FALSE,CycTrigPa:=FALSE,DeadBTransmitPa:=REAL#0.0,TransmitModePa:= INT#1);	Rk10UAct_Q	:=	S_MFI_MNG_368.Analog_Output_Q	;
S_MFI_MNG_369	(MFI_Value:=	emC_LUC[LUC_Num].SCADA.Out.Rk[10].IAct	,TimeTag:=Timestamp,IV:=FALSE,CycTrigPa:=FALSE,DeadBTransmitPa:=REAL#0.0,TransmitModePa:= INT#1);	Rk10IAct_Q	:=	S_MFI_MNG_369.Analog_Output_Q	;
S_MFI_MNG_370	(MFI_Value:=	emC_LUC[LUC_Num].SCADA.Out.Rk[10].TempAct	,TimeTag:=Timestamp,IV:=FALSE,CycTrigPa:=FALSE,DeadBTransmitPa:=REAL#0.0,TransmitModePa:= INT#1);	Rk10TempAct_Q	:=	S_MFI_MNG_370.Analog_Output_Q	;
S_SPI_MNG_371	(Digital_Feedback_Value:=	emC_LUC[LUC_Num].SCADA.Out.Rk[11].OnlineSt	,TimeTag:=Timestamp,IV:=FALSE);	Rk11OnlineSt_Q	:=	S_SPI_MNG_371.Digital_Feedback_Q	;
S_SPI_MNG_372	(Digital_Feedback_Value:=	emC_LUC[LUC_Num].SCADA.Out.Rk[11].FaultSt	,TimeTag:=Timestamp,IV:=FALSE);	Rk11FaultSt_Q	:=	S_SPI_MNG_372.Digital_Feedback_Q	;
S_MFI_MNG_373	(MFI_Value:=	emC_LUC[LUC_Num].SCADA.Out.Rk[11].SoCAct	,TimeTag:=Timestamp,IV:=FALSE,CycTrigPa:=FALSE,DeadBTransmitPa:=REAL#0.0,TransmitModePa:= INT#1);	Rk11SoCAct_Q	:=	S_MFI_MNG_373.Analog_Output_Q	;
S_MFI_MNG_374	(MFI_Value:=	emC_LUC[LUC_Num].SCADA.Out.Rk[11].SoHAct	,TimeTag:=Timestamp,IV:=FALSE,CycTrigPa:=FALSE,DeadBTransmitPa:=REAL#0.0,TransmitModePa:= INT#1);	Rk11SoHAct_Q	:=	S_MFI_MNG_374.Analog_Output_Q	;
S_MFI_MNG_375	(MFI_Value:=	emC_LUC[LUC_Num].SCADA.Out.Rk[11].UAct	,TimeTag:=Timestamp,IV:=FALSE,CycTrigPa:=FALSE,DeadBTransmitPa:=REAL#0.0,TransmitModePa:= INT#1);	Rk11UAct_Q	:=	S_MFI_MNG_375.Analog_Output_Q	;
S_MFI_MNG_376	(MFI_Value:=	emC_LUC[LUC_Num].SCADA.Out.Rk[11].IAct	,TimeTag:=Timestamp,IV:=FALSE,CycTrigPa:=FALSE,DeadBTransmitPa:=REAL#0.0,TransmitModePa:= INT#1);	Rk11IAct_Q	:=	S_MFI_MNG_376.Analog_Output_Q	;
S_MFI_MNG_377	(MFI_Value:=	emC_LUC[LUC_Num].SCADA.Out.Rk[11].TempAct	,TimeTag:=Timestamp,IV:=FALSE,CycTrigPa:=FALSE,DeadBTransmitPa:=REAL#0.0,TransmitModePa:= INT#1);	Rk11TempAct_Q	:=	S_MFI_MNG_377.Analog_Output_Q	;
S_SPI_MNG_378	(Digital_Feedback_Value:=	emC_LUC[LUC_Num].SCADA.Out.Rk[12].OnlineSt	,TimeTag:=Timestamp,IV:=FALSE);	Rk12OnlineSt_Q	:=	S_SPI_MNG_378.Digital_Feedback_Q	;
S_SPI_MNG_379	(Digital_Feedback_Value:=	emC_LUC[LUC_Num].SCADA.Out.Rk[12].FaultSt	,TimeTag:=Timestamp,IV:=FALSE);	Rk12FaultSt_Q	:=	S_SPI_MNG_379.Digital_Feedback_Q	;
S_MFI_MNG_380	(MFI_Value:=	emC_LUC[LUC_Num].SCADA.Out.Rk[12].SoCAct	,TimeTag:=Timestamp,IV:=FALSE,CycTrigPa:=FALSE,DeadBTransmitPa:=REAL#0.0,TransmitModePa:= INT#1);	Rk12SoCAct_Q	:=	S_MFI_MNG_380.Analog_Output_Q	;
S_MFI_MNG_381	(MFI_Value:=	emC_LUC[LUC_Num].SCADA.Out.Rk[12].SoHAct	,TimeTag:=Timestamp,IV:=FALSE,CycTrigPa:=FALSE,DeadBTransmitPa:=REAL#0.0,TransmitModePa:= INT#1);	Rk12SoHAct_Q	:=	S_MFI_MNG_381.Analog_Output_Q	;
S_MFI_MNG_382	(MFI_Value:=	emC_LUC[LUC_Num].SCADA.Out.Rk[12].UAct	,TimeTag:=Timestamp,IV:=FALSE,CycTrigPa:=FALSE,DeadBTransmitPa:=REAL#0.0,TransmitModePa:= INT#1);	Rk12UAct_Q	:=	S_MFI_MNG_382.Analog_Output_Q	;
S_MFI_MNG_383	(MFI_Value:=	emC_LUC[LUC_Num].SCADA.Out.Rk[12].IAct	,TimeTag:=Timestamp,IV:=FALSE,CycTrigPa:=FALSE,DeadBTransmitPa:=REAL#0.0,TransmitModePa:= INT#1);	Rk12IAct_Q	:=	S_MFI_MNG_383.Analog_Output_Q	;
S_MFI_MNG_384	(MFI_Value:=	emC_LUC[LUC_Num].SCADA.Out.Rk[12].TempAct	,TimeTag:=Timestamp,IV:=FALSE,CycTrigPa:=FALSE,DeadBTransmitPa:=REAL#0.0,TransmitModePa:= INT#1);	Rk12TempAct_Q	:=	S_MFI_MNG_384.Analog_Output_Q	;
S_SPI_MNG_385	(Digital_Feedback_Value:=	emC_LUC[LUC_Num].SCADA.Out.Rk[13].OnlineSt	,TimeTag:=Timestamp,IV:=FALSE);	Rk13OnlineSt_Q	:=	S_SPI_MNG_385.Digital_Feedback_Q	;
S_SPI_MNG_386	(Digital_Feedback_Value:=	emC_LUC[LUC_Num].SCADA.Out.Rk[13].FaultSt	,TimeTag:=Timestamp,IV:=FALSE);	Rk13FaultSt_Q	:=	S_SPI_MNG_386.Digital_Feedback_Q	;
S_MFI_MNG_387	(MFI_Value:=	emC_LUC[LUC_Num].SCADA.Out.Rk[13].SoCAct	,TimeTag:=Timestamp,IV:=FALSE,CycTrigPa:=FALSE,DeadBTransmitPa:=REAL#0.0,TransmitModePa:= INT#1);	Rk13SoCAct_Q	:=	S_MFI_MNG_387.Analog_Output_Q	;
S_MFI_MNG_388	(MFI_Value:=	emC_LUC[LUC_Num].SCADA.Out.Rk[13].SoHAct	,TimeTag:=Timestamp,IV:=FALSE,CycTrigPa:=FALSE,DeadBTransmitPa:=REAL#0.0,TransmitModePa:= INT#1);	Rk13SoHAct_Q	:=	S_MFI_MNG_388.Analog_Output_Q	;
S_MFI_MNG_389	(MFI_Value:=	emC_LUC[LUC_Num].SCADA.Out.Rk[13].UAct	,TimeTag:=Timestamp,IV:=FALSE,CycTrigPa:=FALSE,DeadBTransmitPa:=REAL#0.0,TransmitModePa:= INT#1);	Rk13UAct_Q	:=	S_MFI_MNG_389.Analog_Output_Q	;
S_MFI_MNG_390	(MFI_Value:=	emC_LUC[LUC_Num].SCADA.Out.Rk[13].IAct	,TimeTag:=Timestamp,IV:=FALSE,CycTrigPa:=FALSE,DeadBTransmitPa:=REAL#0.0,TransmitModePa:= INT#1);	Rk13IAct_Q	:=	S_MFI_MNG_390.Analog_Output_Q	;
S_MFI_MNG_391	(MFI_Value:=	emC_LUC[LUC_Num].SCADA.Out.Rk[13].TempAct	,TimeTag:=Timestamp,IV:=FALSE,CycTrigPa:=FALSE,DeadBTransmitPa:=REAL#0.0,TransmitModePa:= INT#1);	Rk13TempAct_Q	:=	S_MFI_MNG_391.Analog_Output_Q	;
S_SPI_MNG_392	(Digital_Feedback_Value:=	emC_LUC[LUC_Num].SCADA.Out.Rk[14].OnlineSt	,TimeTag:=Timestamp,IV:=FALSE);	Rk14OnlineSt_Q	:=	S_SPI_MNG_392.Digital_Feedback_Q	;
S_SPI_MNG_393	(Digital_Feedback_Value:=	emC_LUC[LUC_Num].SCADA.Out.Rk[14].FaultSt	,TimeTag:=Timestamp,IV:=FALSE);	Rk14FaultSt_Q	:=	S_SPI_MNG_393.Digital_Feedback_Q	;
S_MFI_MNG_394	(MFI_Value:=	emC_LUC[LUC_Num].SCADA.Out.Rk[14].SoCAct	,TimeTag:=Timestamp,IV:=FALSE,CycTrigPa:=FALSE,DeadBTransmitPa:=REAL#0.0,TransmitModePa:= INT#1);	Rk14SoCAct_Q	:=	S_MFI_MNG_394.Analog_Output_Q	;
S_MFI_MNG_395	(MFI_Value:=	emC_LUC[LUC_Num].SCADA.Out.Rk[14].SoHAct	,TimeTag:=Timestamp,IV:=FALSE,CycTrigPa:=FALSE,DeadBTransmitPa:=REAL#0.0,TransmitModePa:= INT#1);	Rk14SoHAct_Q	:=	S_MFI_MNG_395.Analog_Output_Q	;
S_MFI_MNG_396	(MFI_Value:=	emC_LUC[LUC_Num].SCADA.Out.Rk[14].UAct	,TimeTag:=Timestamp,IV:=FALSE,CycTrigPa:=FALSE,DeadBTransmitPa:=REAL#0.0,TransmitModePa:= INT#1);	Rk14UAct_Q	:=	S_MFI_MNG_396.Analog_Output_Q	;
S_MFI_MNG_397	(MFI_Value:=	emC_LUC[LUC_Num].SCADA.Out.Rk[14].IAct	,TimeTag:=Timestamp,IV:=FALSE,CycTrigPa:=FALSE,DeadBTransmitPa:=REAL#0.0,TransmitModePa:= INT#1);	Rk14IAct_Q	:=	S_MFI_MNG_397.Analog_Output_Q	;
S_MFI_MNG_398	(MFI_Value:=	emC_LUC[LUC_Num].SCADA.Out.Rk[14].TempAct	,TimeTag:=Timestamp,IV:=FALSE,CycTrigPa:=FALSE,DeadBTransmitPa:=REAL#0.0,TransmitModePa:= INT#1);	Rk14TempAct_Q	:=	S_MFI_MNG_398.Analog_Output_Q	;
S_SPI_MNG_399	(Digital_Feedback_Value:=	emC_LUC[LUC_Num].SCADA.Out.Rk[15].OnlineSt	,TimeTag:=Timestamp,IV:=FALSE);	Rk15OnlineSt_Q	:=	S_SPI_MNG_399.Digital_Feedback_Q	;
S_SPI_MNG_400	(Digital_Feedback_Value:=	emC_LUC[LUC_Num].SCADA.Out.Rk[15].FaultSt	,TimeTag:=Timestamp,IV:=FALSE);	Rk15FaultSt_Q	:=	S_SPI_MNG_400.Digital_Feedback_Q	;
S_MFI_MNG_401	(MFI_Value:=	emC_LUC[LUC_Num].SCADA.Out.Rk[15].SoCAct	,TimeTag:=Timestamp,IV:=FALSE,CycTrigPa:=FALSE,DeadBTransmitPa:=REAL#0.0,TransmitModePa:= INT#1);	Rk15SoCAct_Q	:=	S_MFI_MNG_401.Analog_Output_Q	;
S_MFI_MNG_402	(MFI_Value:=	emC_LUC[LUC_Num].SCADA.Out.Rk[15].SoHAct	,TimeTag:=Timestamp,IV:=FALSE,CycTrigPa:=FALSE,DeadBTransmitPa:=REAL#0.0,TransmitModePa:= INT#1);	Rk15SoHAct_Q	:=	S_MFI_MNG_402.Analog_Output_Q	;
S_MFI_MNG_403	(MFI_Value:=	emC_LUC[LUC_Num].SCADA.Out.Rk[15].UAct	,TimeTag:=Timestamp,IV:=FALSE,CycTrigPa:=FALSE,DeadBTransmitPa:=REAL#0.0,TransmitModePa:= INT#1);	Rk15UAct_Q	:=	S_MFI_MNG_403.Analog_Output_Q	;
S_MFI_MNG_404	(MFI_Value:=	emC_LUC[LUC_Num].SCADA.Out.Rk[15].IAct	,TimeTag:=Timestamp,IV:=FALSE,CycTrigPa:=FALSE,DeadBTransmitPa:=REAL#0.0,TransmitModePa:= INT#1);	Rk15IAct_Q	:=	S_MFI_MNG_404.Analog_Output_Q	;
S_MFI_MNG_405	(MFI_Value:=	emC_LUC[LUC_Num].SCADA.Out.Rk[15].TempAct	,TimeTag:=Timestamp,IV:=FALSE,CycTrigPa:=FALSE,DeadBTransmitPa:=REAL#0.0,TransmitModePa:= INT#1);	Rk15TempAct_Q	:=	S_MFI_MNG_405.Analog_Output_Q	;
S_SPI_MNG_406	(Digital_Feedback_Value:=	emC_LUC[LUC_Num].SCADA.Out.Rk[16].OnlineSt	,TimeTag:=Timestamp,IV:=FALSE);	Rk16OnlineSt_Q	:=	S_SPI_MNG_406.Digital_Feedback_Q	;
S_SPI_MNG_407	(Digital_Feedback_Value:=	emC_LUC[LUC_Num].SCADA.Out.Rk[16].FaultSt	,TimeTag:=Timestamp,IV:=FALSE);	Rk16FaultSt_Q	:=	S_SPI_MNG_407.Digital_Feedback_Q	;
S_MFI_MNG_408	(MFI_Value:=	emC_LUC[LUC_Num].SCADA.Out.Rk[16].SoCAct	,TimeTag:=Timestamp,IV:=FALSE,CycTrigPa:=FALSE,DeadBTransmitPa:=REAL#0.0,TransmitModePa:= INT#1);	Rk16SoCAct_Q	:=	S_MFI_MNG_408.Analog_Output_Q	;
S_MFI_MNG_409	(MFI_Value:=	emC_LUC[LUC_Num].SCADA.Out.Rk[16].SoHAct	,TimeTag:=Timestamp,IV:=FALSE,CycTrigPa:=FALSE,DeadBTransmitPa:=REAL#0.0,TransmitModePa:= INT#1);	Rk16SoHAct_Q	:=	S_MFI_MNG_409.Analog_Output_Q	;
S_MFI_MNG_410	(MFI_Value:=	emC_LUC[LUC_Num].SCADA.Out.Rk[16].UAct	,TimeTag:=Timestamp,IV:=FALSE,CycTrigPa:=FALSE,DeadBTransmitPa:=REAL#0.0,TransmitModePa:= INT#1);	Rk16UAct_Q	:=	S_MFI_MNG_410.Analog_Output_Q	;
S_MFI_MNG_411	(MFI_Value:=	emC_LUC[LUC_Num].SCADA.Out.Rk[16].IAct	,TimeTag:=Timestamp,IV:=FALSE,CycTrigPa:=FALSE,DeadBTransmitPa:=REAL#0.0,TransmitModePa:= INT#1);	Rk16IAct_Q	:=	S_MFI_MNG_411.Analog_Output_Q	;
S_MFI_MNG_412	(MFI_Value:=	emC_LUC[LUC_Num].SCADA.Out.Rk[16].TempAct	,TimeTag:=Timestamp,IV:=FALSE,CycTrigPa:=FALSE,DeadBTransmitPa:=REAL#0.0,TransmitModePa:= INT#1);	Rk16TempAct_Q	:=	S_MFI_MNG_412.Analog_Output_Q	;
S_SPI_MNG_413	(Digital_Feedback_Value:=	emC_LUC[LUC_Num].SCADA.Out.Rk[17].OnlineSt	,TimeTag:=Timestamp,IV:=FALSE);	Rk17OnlineSt_Q	:=	S_SPI_MNG_413.Digital_Feedback_Q	;
S_SPI_MNG_414	(Digital_Feedback_Value:=	emC_LUC[LUC_Num].SCADA.Out.Rk[17].FaultSt	,TimeTag:=Timestamp,IV:=FALSE);	Rk17FaultSt_Q	:=	S_SPI_MNG_414.Digital_Feedback_Q	;
S_MFI_MNG_415	(MFI_Value:=	emC_LUC[LUC_Num].SCADA.Out.Rk[17].SoCAct	,TimeTag:=Timestamp,IV:=FALSE,CycTrigPa:=FALSE,DeadBTransmitPa:=REAL#0.0,TransmitModePa:= INT#1);	Rk17SoCAct_Q	:=	S_MFI_MNG_415.Analog_Output_Q	;
S_MFI_MNG_416	(MFI_Value:=	emC_LUC[LUC_Num].SCADA.Out.Rk[17].SoHAct	,TimeTag:=Timestamp,IV:=FALSE,CycTrigPa:=FALSE,DeadBTransmitPa:=REAL#0.0,TransmitModePa:= INT#1);	Rk17SoHAct_Q	:=	S_MFI_MNG_416.Analog_Output_Q	;
S_MFI_MNG_417	(MFI_Value:=	emC_LUC[LUC_Num].SCADA.Out.Rk[17].UAct	,TimeTag:=Timestamp,IV:=FALSE,CycTrigPa:=FALSE,DeadBTransmitPa:=REAL#0.0,TransmitModePa:= INT#1);	Rk17UAct_Q	:=	S_MFI_MNG_417.Analog_Output_Q	;
S_MFI_MNG_418	(MFI_Value:=	emC_LUC[LUC_Num].SCADA.Out.Rk[17].IAct	,TimeTag:=Timestamp,IV:=FALSE,CycTrigPa:=FALSE,DeadBTransmitPa:=REAL#0.0,TransmitModePa:= INT#1);	Rk17IAct_Q	:=	S_MFI_MNG_418.Analog_Output_Q	;
S_MFI_MNG_419	(MFI_Value:=	emC_LUC[LUC_Num].SCADA.Out.Rk[17].TempAct	,TimeTag:=Timestamp,IV:=FALSE,CycTrigPa:=FALSE,DeadBTransmitPa:=REAL#0.0,TransmitModePa:= INT#1);	Rk17TempAct_Q	:=	S_MFI_MNG_419.Analog_Output_Q	;
S_SPI_MNG_420	(Digital_Feedback_Value:=	emC_LUC[LUC_Num].SCADA.Out.Rk[18].OnlineSt	,TimeTag:=Timestamp,IV:=FALSE);	Rk18OnlineSt_Q	:=	S_SPI_MNG_420.Digital_Feedback_Q	;
S_SPI_MNG_421	(Digital_Feedback_Value:=	emC_LUC[LUC_Num].SCADA.Out.Rk[18].FaultSt	,TimeTag:=Timestamp,IV:=FALSE);	Rk18FaultSt_Q	:=	S_SPI_MNG_421.Digital_Feedback_Q	;
S_MFI_MNG_422	(MFI_Value:=	emC_LUC[LUC_Num].SCADA.Out.Rk[18].SoCAct	,TimeTag:=Timestamp,IV:=FALSE,CycTrigPa:=FALSE,DeadBTransmitPa:=REAL#0.0,TransmitModePa:= INT#1);	Rk18SoCAct_Q	:=	S_MFI_MNG_422.Analog_Output_Q	;
S_MFI_MNG_423	(MFI_Value:=	emC_LUC[LUC_Num].SCADA.Out.Rk[18].SoHAct	,TimeTag:=Timestamp,IV:=FALSE,CycTrigPa:=FALSE,DeadBTransmitPa:=REAL#0.0,TransmitModePa:= INT#1);	Rk18SoHAct_Q	:=	S_MFI_MNG_423.Analog_Output_Q	;
S_MFI_MNG_424	(MFI_Value:=	emC_LUC[LUC_Num].SCADA.Out.Rk[18].UAct	,TimeTag:=Timestamp,IV:=FALSE,CycTrigPa:=FALSE,DeadBTransmitPa:=REAL#0.0,TransmitModePa:= INT#1);	Rk18UAct_Q	:=	S_MFI_MNG_424.Analog_Output_Q	;
S_MFI_MNG_425	(MFI_Value:=	emC_LUC[LUC_Num].SCADA.Out.Rk[18].IAct	,TimeTag:=Timestamp,IV:=FALSE,CycTrigPa:=FALSE,DeadBTransmitPa:=REAL#0.0,TransmitModePa:= INT#1);	Rk18IAct_Q	:=	S_MFI_MNG_425.Analog_Output_Q	;
S_MFI_MNG_426	(MFI_Value:=	emC_LUC[LUC_Num].SCADA.Out.Rk[18].TempAct	,TimeTag:=Timestamp,IV:=FALSE,CycTrigPa:=FALSE,DeadBTransmitPa:=REAL#0.0,TransmitModePa:= INT#1);	Rk18TempAct_Q	:=	S_MFI_MNG_426.Analog_Output_Q	;
							
							emC_LUC[LUC_Num].PPC.PPCOut.GCFaultSt	:=	emC_LUC[LUC_Num].emPs.PS.GCFaultSt	;
emC_LUC[LUC_Num].PPC.PPCOut.NonCriticalAlarm	:=	emC_LUC[LUC_Num].SM.In.NonCriticalAlarm	;
emC_LUC[LUC_Num].PPC.PPCOut.CriticalAlarm	:=	emC_LUC[LUC_Num].SM.In.CriticalAlarm	;
emC_LUC[LUC_Num].PPC.PPCOut.Warning	:=	emC_LUC[LUC_Num].SM.In.Warning	;
emC_LUC[LUC_Num].PPC.PPCOut.StoppingSt	:=	emC_LUC[LUC_Num].SM.Out.StoppingSt	;
emC_LUC[LUC_Num].PPC.PPCOut.CtrlSystemReady	:=	emC_LUC[LUC_Num].emPs.PS.CtrlSystemReady	;
emC_LUC[LUC_Num].PPC.PPCOut.OnlineSt	:=	emC_LUC[LUC_Num].SM.In.OnlineSt	;
emC_LUC[LUC_Num].PPC.PPCOut.RunningSt	:=	emC_LUC[LUC_Num].SM.In.RunningSt	;
								
								
emC_LUC[LUC_Num].PPC.PPCOut.TempAct	:=	emC_LUC[LUC_Num].emPs.PS.TempAct  		;
emC_LUC[LUC_Num].PPC.PPCOut.BatPNomMaxAct	:=	emC_LUC[LUC_Num].BattPLC.CtrlLo.Out.Batt_Sys.BattSysMeasure.BatPNomMaxAct  		;
emC_LUC[LUC_Num].PPC.PPCOut.BatPNomMinAct	:=	emC_LUC[LUC_Num].BattPLC.CtrlLo.Out.Batt_Sys.BattSysMeasure.BatPNomMinAct  		;
emC_LUC[LUC_Num].PPC.PPCOut.SocPctAct	:=	emC_LUC[LUC_Num].BattPLC.CtrlLo.Out.Batt_Sys.BattSysMeasure.SocPctAct  		;
emC_LUC[LUC_Num].PPC.PPCOut.UAct	:=	emC_LUC[LUC_Num].emPs.PS.GCUAct  		;
emC_LUC[LUC_Num].PPC.PPCOut.FAct	:=	emC_LUC[LUC_Num].emPs.PS.GCFAct  		;
emC_LUC[LUC_Num].PPC.PPCOut.PAct	:=	emC_LUC[LUC_Num].emPs.PS.GCPAct  		;
emC_LUC[LUC_Num].PPC.PPCOut.QAct	:=	emC_LUC[LUC_Num].emPs.PS.GCQAct  		;
								
								
emC_PPCOut_1(									
				GCFaultSt		:=	emC_LUC[LUC_Num].PPC.PPCOut.GCFaultSt	,	
				NonCriticalAlarm		:=	emC_LUC[LUC_Num].PPC.PPCOut.NonCriticalAlarm	,	
				CriticalAlarm		:=	emC_LUC[LUC_Num].PPC.PPCOut.CriticalAlarm	,	
				Warning		:=	emC_LUC[LUC_Num].PPC.PPCOut.Warning	,	
				StoppingSt		:=	emC_LUC[LUC_Num].PPC.PPCOut.StoppingSt	,	
				CtrlSystemReady		:=	emC_LUC[LUC_Num].PPC.PPCOut.CtrlSystemReady	,
				BlackSys	:=	emC_LUC[LUC_Num].PPC.PPCOut.BlackSys	,	
				OnlineSt		:=	emC_LUC[LUC_Num].PPC.PPCOut.OnlineSt	,	
				RunningSt		:=	emC_LUC[LUC_Num].PPC.PPCOut.RunningSt	,	
				TempAct		:=	emC_LUC[LUC_Num].PPC.PPCOut.TempAct	,	
				BatPNomMaxAct		:=	emC_LUC[LUC_Num].PPC.PPCOut.BatPNomMaxAct	,	
				BatPNomMinAct		:=	emC_LUC[LUC_Num].PPC.PPCOut.BatPNomMinAct	,	
				SocPctAct		:=	emC_LUC[LUC_Num].PPC.PPCOut.SocPctAct	,	
				UAct		:=	emC_LUC[LUC_Num].PPC.PPCOut.UAct	,	
				FAct		:=	emC_LUC[LUC_Num].PPC.PPCOut.FAct	,	
				PAct		:=	emC_LUC[LUC_Num].PPC.PPCOut.PAct	,	
				QAct		:=	emC_LUC[LUC_Num].PPC.PPCOut.QAct	,	
				Timestamp		:=	 Timestamp	)	;
	PPC_GCFaultSt_Q	:=	emC_PPCOut_1.PPC_GCFaultSt_Q	;					
	PPC_NonCriticalAl_Q	:=	emC_PPCOut_1.PPC_NonCriticalAl_Q	;					
	PPC_CriticalAl_Q	:=	emC_PPCOut_1.PPC_CriticalAl_Q	;					
	PPC_WarningAl_Q	:=	emC_PPCOut_1.PPC_WarningAl_Q	;					
	PPC_StoppingSt_Q	:=	emC_PPCOut_1.PPC_StoppingSt_Q	;					
	PPC_CtrlSystemReady_Q	:=	emC_PPCOut_1.PPC_CtrlSystemReady_Q	;					
	PPC_BlackSys_Q	:=	emC_PPCOut_1.PPC_BlackSys_Q	;					
	PPC_OnlineSt_Q	:=	emC_PPCOut_1.PPC_OnlineSt_Q	;					
	PPC_RunningSt_Q	:=	emC_PPCOut_1.PPC_RunningSt_Q	;					
	PPC_TempAct_Q	:=	emC_PPCOut_1.PPC_TempAct_Q	;					
	PPC_BatPNomMaxAct_Q	:=	emC_PPCOut_1.PPC_BatPNomMaxAct_Q	;					
	PPC_BatPNomMinAct_Q	:=	emC_PPCOut_1.PPC_BatPNomMinAct_Q	;					
	PPC_BatSocAct_Q	:=	emC_PPCOut_1.PPC_BatSocAct_Q	;					
	PPC_UAct_Q	:=	emC_PPCOut_1.PPC_UAct_Q	;					
	PPC_FAct_Q	:=	emC_PPCOut_1.PPC_FAct_Q	;					
	PPC_PAct_Q	:=	emC_PPCOut_1.PPC_PAct_Q	;					
	PPC_QAct_Q	:=	emC_PPCOut_1.PPC_QAct_Q	;
							
						
					
END_PROGRAM

PROGRAM emCBSSim01_Fed01
  VAR
    Fed_MG_1 : Fed_MG;
  END_VAR
  VAR_EXTERNAL
    Fed_Data : Feeder_Data;
    Sys_Data : Sys_Data;
    TStep : TIME;
    HMIFeeder_Var_IN : Feeder_Var_IN;
  END_VAR

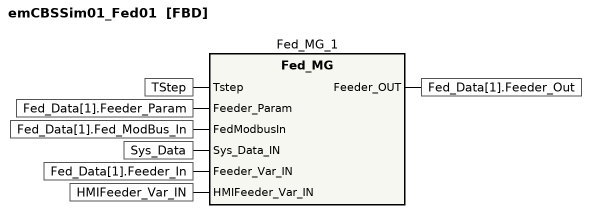
(* FBD diagram, written out as Structured Text *)
Fed_MG_1(Tstep := TStep, Feeder_Param := Fed_Data[1].Feeder_Param, FedModbusIn := Fed_Data[1].Fed_ModBus_In, Sys_Data_IN := Sys_Data, Feeder_Var_IN := Fed_Data[1].Feeder_In, HMIFeeder_Var_IN := HMIFeeder_Var_IN);
Fed_Data[1].Feeder_Out := Fed_MG_1.Feeder_OUT;
END_PROGRAM

PROGRAM emCBSSim01_Grid01
  VAR
    GridSim_1 : GridSim;
    PLCCycle_1 : PLCCycle;
  END_VAR
  VAR_EXTERNAL
    TStep : TIME;
    PLC_TICKS_PER_SEC : INT;
    Grid_Dat : Grid_Dat;
    Sys_Data : Sys_Data;
  END_VAR
  VAR
    Synch_MG_1_1 : Synch_MG_1;
  END_VAR
  VAR_EXTERNAL
    Synch_Parameters : Synch_Parameters;
  END_VAR
  VAR
    Grid_Sum_1 : Grid_Sum;
  END_VAR
  VAR_EXTERNAL
    PS : Ps_LineUP;
    LuNumPa : INT;
  END_VAR
  VAR
    StartSynching : BOOL;
    BreakerCloseCmd : BOOL;
    SyncCheckSt : BOOL;
  END_VAR

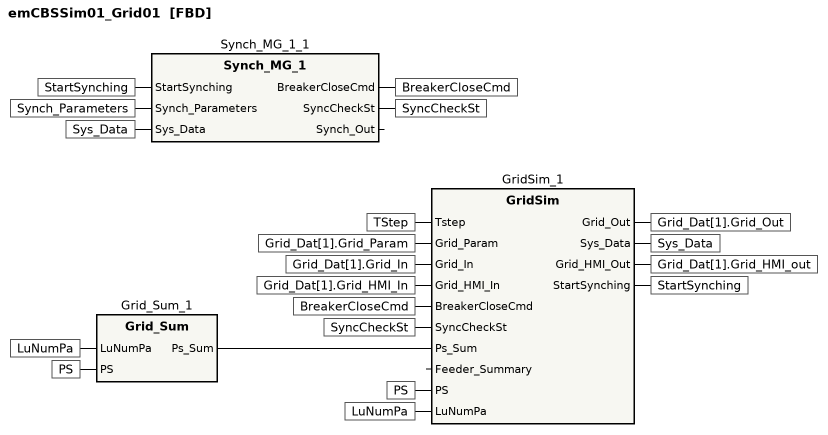
(* FBD diagram, written out as Structured Text *)
Grid_Sum_1(LuNumPa := LuNumPa, PS := PS);
GridSim_1(Tstep := TStep, Grid_Param := Grid_Dat[1].Grid_Param, Grid_In := Grid_Dat[1].Grid_In, Grid_HMI_In := Grid_Dat[1].Grid_HMI_In, BreakerCloseCmd := BreakerCloseCmd, SyncCheckSt := SyncCheckSt, Ps_Sum := Grid_Sum_1.Ps_Sum, PS := PS, LuNumPa := LuNumPa);
Grid_Dat[1].Grid_Out := GridSim_1.Grid_Out;
Sys_Data := GridSim_1.Sys_Data;
Grid_Dat[1].Grid_HMI_out := GridSim_1.Grid_HMI_Out;
StartSynching := GridSim_1.StartSynching;
Synch_MG_1_1(StartSynching := StartSynching, Synch_Parameters := Synch_Parameters, Sys_Data := Sys_Data);
SyncCheckSt := Synch_MG_1_1.SyncCheckSt;
BreakerCloseCmd := Synch_MG_1_1.BreakerCloseCmd;
END_PROGRAM

PROGRAM emCBSSim01_In
  VAR
    BMS_Cmd_In_I : TDC;
    BMS_Cmd_In_Q : TDC;
    BMS_Cmd_Rsp_Q : TDC;
  END_VAR
  VAR_EXTERNAL
    Sys_Parameters : Sys_Parameters;
    Grid_Dat : Grid_Dat;
  END_VAR
  VAR
    PS_Var_In : PS_Var_In;
  END_VAR
  VAR_EXTERNAL
    Synch_Parameters : Synch_Parameters;
  END_VAR
  VAR
    Grid_Modbus_In_1 : Grid_Modbus_In;
    Fed_ModInBlock_1 : Fed_ModInBlock;
    Grid_01_CloseCmd_I : SCO;
    Grid_01_OpenCmd_I : SCO;
    Grid_01_AlarmReset_I : SCO;
    Grid_01_AlarmReset_Q : SCO;
    Grid_01_OpenCmd_Q : SCO;
    Grid_01_CloseCmd_Q : SCO;
    Fed_01_CloseCmd_Q : SCO;
    Fed_01_OpenCmd_Q : SCO;
    Fed_01_AlarmReset_Q : SCO;
    Fed_01_AlarmReset_I : SCO;
    Fed_01_OpenCmd_I : SCO;
    Fed_01_CloseCmd_I : SCO;
  END_VAR
  VAR_EXTERNAL
    Fed_Data : Feeder_Data;
  END_VAR
  VAR
    Grid_Var_In_1 : Grid_HMI_Var_In;
    Fed_Var_In_1 : Fed_Var_In;
    PS_Var_In_1 : PS_Var_In;
    PS_Var_In_2 : PS_Var_In;
    PS_Var_In_3 : PS_Var_In;
    PS_Var_In_4 : PS_Var_In;
    PS_Var_In_5 : PS_Var_In;
    PS1_GcStartCmd_S : BOOL;
    PS1_GcStopCmd_S : BOOL;
    GcBreakerCloseCmd_S : BOOL;
    PS1_GcBreakerCloseCmd_S : BOOL;
    PS1_GcBreakerOpenCmd_S : BOOL;
    PS1_GcAlarmReset_S : BOOL;
    PS1_GcSim_CritAl_S : BOOL;
    PS1_GcSim_NonCritAl_S : BOOL;
    PS1_GcSim_WarnAl_S : BOOL;
    PS1_GcEStop_S : BOOL;
    PS1_BattStartCmd_S : BOOL;
    PS1_BattStopCmd_S : BOOL;
    PS1_BattAlarmReset_S : BOOL;
    PS1_BattSim_CritAl_S : BOOL;
    PS1_BattSim_NonCritAl_S : BOOL;
    PS1_BattSim_WarnAl_S : BOOL;
    PS1_BattEStop_S : BOOL;
    PS1_BattSim_FireAl_S : BOOL;
    PS1_Rk1InService_S : BOOL := TRUE;
    PS1_Rk1RkCloseCmd_S : BOOL;
    PS1_Rk1RkOpenCmd_S : BOOL;
    PS1_Rk1RkAlarm_S : BOOL;
    PS1_Rk2InService_S : BOOL := TRUE;
    PS1_Rk2RkCloseCmd_S : BOOL;
    PS1_Rk2RkOpenCmd_S : BOOL;
    PS1_Rk2RkAlarm_S : BOOL;
    PS1_Rk3InService_S : BOOL := TRUE;
    PS1_Rk3RkCloseCmd_S : BOOL;
    PS1_Rk3RkOpenCmd_S : BOOL;
    PS1_Rk3RkAlarm_S : BOOL;
    PS1_Rk4InService_S : BOOL := TRUE;
    PS1_Rk4RkCloseCmd_S : BOOL;
    PS1_Rk4RkOpenCmd_S : BOOL;
    PS1_Rk4RkAlarm_S : BOOL;
    PS1_Rk5InService_S : BOOL := TRUE;
    PS1_Rk5RkCloseCmd_S : BOOL;
    PS1_Rk5RkOpenCmd_S : BOOL;
    PS1_Rk5RkAlarm_S : BOOL;
    LuNumPa_S : INT := 5;
  END_VAR
  VAR_EXTERNAL
    LuNumPa : INT;
  END_VAR
  VAR
    Grid_Param_In_1 : Grid_Param_In;
    Fed_Var_In_2 : Fed_Var_In;
  END_VAR
  VAR_EXTERNAL
    HMIFeeder_Var_IN : Feeder_Var_IN;
  END_VAR
  VAR
    Grid_HMI_Var_In_1 : Grid_HMI_Var_In;
    BattTotalRackCntPa_S : USINT := 5;
    BattPartMinRackCntPa_S : USINT := 4;
    Ps_Sim_Param_1 : Ps_Sim_Param;
    Ps_Sim_Param_2 : Ps_Sim_Param;
    Ps_Sim_Param_3 : Ps_Sim_Param;
    Ps_Sim_Param_4 : Ps_Sim_Param;
    Ps_Sim_Param_5 : Ps_Sim_Param;
  END_VAR
  VAR_EXTERNAL
    PS : Ps_LineUP;
  END_VAR
  VAR
    Gc_PQ_FU_RefSelPa_S : INT := 2;
    Gc_FNomPa_S : REAL := 50.0;
    Gc_UNomPa_S : REAL := 480.0;
    Gc_SNomPa_S : REAL := 1000.0;
    Gc_fDroopPa_S : REAL := 0.01;
    Gc_UDroopPa_S : REAL := 0.01;
    Gc_TMotorPa_S : TIME := T#1.5s;
    Gc_TExciterPa_S : TIME := T#0.05s;
    Gc_P_UpPa_S : REAL := 50.0;
    Gc_P_DownPa_S : REAL := 50.0;
    Gc_PLimMinPa_S : REAL := -1000.0;
    Gc_PLimMaxPa_S : REAL := 1000.0;
    Gc_PinitPa_S : REAL := 0.0;
    Gc_PNomPa_S : REAL := 1000.0;
    Gc_QLimMinPa_S : REAL := -300.0;
    Gc_QLimMaxPa_S : REAL := 300.0;
    Gc_QinitPa_S : REAL := 0.0;
    Gc_QNomPa_S : REAL := 300.0;
    Gc_OvPFactorPa_S : REAL := 1.5;
    Gc_OvPLockInTPa_S : TIME := T#10s;
    Gc_OvQFactorPa_S : REAL := 1.5;
    Gc_OvQLockInTPa_S : TIME := T#10s;
    Gc_OvUFactorPa_S : REAL := 1.5;
    Gc_OvULockInTPa_S : TIME := T#10s;
    Gc_OvFFactorPa_S : REAL := 1.5;
    Gc_OvFLockInTPa_S : TIME := T#10s;
    BatUNomPa_S : REAL := 700.0;
    BatSNomPa_S : REAL := 1000.0;
    BatEInitPa_S : REAL := 500.0;
    BatENomPa_S : REAL := 1000.0;
    BatEnDerateWrtSocPa_S : BOOL := 0;
    BatEnDerateWrtTempPa_S : BOOL := 0;
    BatDrtChrgOnSocLookUpSocPa : DerateLookUp;
    BatDrtChrgOnSocLookUpDrtPa : DerateLookUp;
    BatDrtDChrgOnSocLookUpSocPa : DerateLookUp;
    BatDrtDChrgOnSocLookUpDrtPa : DerateLookUp;
    BatDerateTempLookUpTempPa : DerateLookUp;
    BatDerateTempLookUpDeratePa : DerateLookUp;
    BatPNomMinPa_S : REAL := -1000.0;
    BatPNomMaxPa_S : REAL := 1000.0;
    BatUMaxPa_S : REAL := 810.0;
    BatUMinPa_S : REAL := 600.0;
    BMSModbus_In_1 : BMSModbus_In;
    BMSModbus_In_2 : BMSModbus_In;
    BMSModbus_In_3 : BMSModbus_In;
    BMSModbus_In_4 : BMSModbus_In;
    BMSModbus_In_5 : BMSModbus_In;
    Fed_Param_In_1 : Fed_Param_In;
    PSModbus_In_1 : PSModbus_In;
    PSModbus_In_2 : PSModbus_In;
    PSModbus_In_3 : PSModbus_In;
    PSModbus_In_4 : PSModbus_In;
    PSModbus_In_5 : PSModbus_In;
    TDC_Cmd_In : TDC;
    TDC_Cmd_Out : TDC;
    TDC_Mon_Out : TDC;
    L1_Gc_Cmd_In_I : TDC;
    L1_Gc_Cmd_In_Q : TDC;
    L1_Gc_Cmd_Rsp_Q : TDC;
    L1_BMS_Cmd_In_Q : TDC;
    L1_BMS_Cmd_Rsp_Q : TDC;
    L1_BMS_Cmd_In_I : TDC;
    L2_Gc_Cmd_In_I : TDC;
    L2_Gc_Cmd_In_Q : TDC;
    L2_Gc_Cmd_Rsp_Q : TDC;
    L2_BMS_Cmd_In_Q : TDC;
    L2_BMS_Cmd_Rsp_Q : TDC;
    L2_BMS_Cmd_In_I : TDC;
    L3_Gc_Cmd_In_I : TDC;
    L3_Gc_Cmd_In_Q : TDC;
    L3_Gc_Cmd_Rsp_Q : TDC;
    L3_BMS_Cmd_In_Q : TDC;
    L3_BMS_Cmd_Rsp_Q : TDC;
    L3_BMS_Cmd_In_I : TDC;
    L4_Gc_Cmd_In_I : TDC;
    L4_Gc_Cmd_In_Q : TDC;
    L4_Gc_Cmd_Rsp_Q : TDC;
    L4_BMS_Cmd_In_Q : TDC;
    L4_BMS_Cmd_Rsp_Q : TDC;
    L4_BMS_Cmd_In_I : TDC;
    L5_Gc_Cmd_In_I : TDC;
    L5_Gc_Cmd_In_Q : TDC;
    L5_Gc_Cmd_Rsp_Q : TDC;
    L5_BMS_Cmd_In_Q : TDC;
    L5_BMS_Cmd_Rsp_Q : TDC;
    L5_BMS_Cmd_In_I : TDC;
  END_VAR

						
							LuNumPa := LuNumPa_S;
(*___________________________________________________________*)
(*Grid*)
Grid_Param_In_1();
Grid_Dat[1].Grid_Param	:=Grid_Param_In_1.Grid_Param;
Sys_Parameters		:=Grid_Param_In_1.Sys_Parameters;
Synch_Parameters	:=Grid_Param_In_1.Synch_Parameters;
(*___________________________________________________________*)
(*Feeder*)
Fed_Param_In_1();
Fed_Data[1].Feeder_Param   :=Fed_Param_In_1.Feeder_Param;
Fed_Var_In_2();
HMIFeeder_Var_IN:=Fed_Var_In_2.Feeder_Var_IN;
								
								
(*___________________________________________________________*)
(*Line Up 1*)
								
Ps_Sim_Param_1(										
				Gc_PQ_FU_RefSelPa_S	:=	Gc_PQ_FU_RefSelPa_S		(* INT *),			
				Gc_SNomPa_S	:=	Gc_SNomPa_S		(* REAL *),		
				Gc_fDroopPa_S	:=	Gc_fDroopPa_S		(* REAL *),		
				Gc_UDroopPa_S	:=	Gc_UDroopPa_S		(* REAL *),		
				Gc_TMotorPa_S	:=	Gc_TMotorPa_S		(* TIME *),		
				Gc_TExciterPa_S	:=	Gc_TExciterPa_S		(* TIME *),		
				Gc_P_UpPa_S	:=	Gc_P_UpPa_S		(* REAL *),		
				Gc_P_DownPa_S	:=	Gc_P_DownPa_S		(* REAL *),		
				Gc_PLimMinPa_S	:=	Gc_PLimMinPa_S		(* REAL *),		
				Gc_PLimMaxPa_S	:=	Gc_PLimMaxPa_S		(* REAL *),		
				Gc_PinitPa_S	:=	Gc_PinitPa_S		(* REAL *),		
				Gc_PNomPa_S	:=	Gc_PNomPa_S		(* REAL *),		
				Gc_QLimMinPa_S	:=	Gc_QLimMinPa_S		(* REAL *),		
				Gc_QLimMaxPa_S	:=	Gc_QLimMaxPa_S		(* REAL *),		
				Gc_QinitPa_S	:=	Gc_QinitPa_S		(* REAL *),		
				Gc_QNomPa_S	:=	Gc_QNomPa_S		(* REAL *),		
				Gc_OvPFactorPa_S	:=	Gc_OvPFactorPa_S		(* REAL *),		
				Gc_OvPLockInTPa_S	:=	Gc_OvPLockInTPa_S		(* TIME *),		
				Gc_OvQFactorPa_S	:=	Gc_OvQFactorPa_S		(* REAL *),		
				Gc_OvQLockInTPa_S	:=	Gc_OvQLockInTPa_S		(* TIME *),		
				Gc_OvUFactorPa_S	:=	Gc_OvUFactorPa_S		(* REAL *),		
				Gc_OvULockInTPa_S	:=	Gc_OvULockInTPa_S		(* TIME *),		
				Gc_OvFFactorPa_S	:=	Gc_OvFFactorPa_S		(* REAL *),		
				Gc_OvFLockInTPa_S	:=	Gc_OvFLockInTPa_S		(* TIME *),		
				BatUNomPa_S	:=	BatUNomPa_S		(* REAL *),		
				BatSNomPa_S	:=	BatSNomPa_S		(* REAL *),		
				BatEInitPa_S	:=	BatEInitPa_S		(* REAL *),		
				BatENomPa_S	:=	BatENomPa_S		(* REAL *),		
				BatEnDerateWrtSocPa_S	:=	BatEnDerateWrtSocPa_S		(* BOOL *),		
				BatEnDerateWrtTempPa_S	:=	BatEnDerateWrtTempPa_S		(* BOOL *),		
				BatDrtChrgOnSocLookUpSocPa	:=	BatDrtChrgOnSocLookUpSocPa		(* DerateLookUp *),		
				BatDrtChrgOnSocLookUpDrtPa	:=	BatDrtChrgOnSocLookUpDrtPa		(* DerateLookUp *),		
				BatDrtDChrgOnSocLookUpSocPa	:=	BatDrtDChrgOnSocLookUpSocPa		(* DerateLookUp *),		
				BatDrtDChrgOnSocLookUpDrtPa	:=	BatDrtDChrgOnSocLookUpDrtPa		(* DerateLookUp *),		
				BatDerateTempLookUpTempPa	:=	BatDerateTempLookUpTempPa		(* DerateLookUp *),		
				BatDerateTempLookUpDeratePa	:=	BatDerateTempLookUpDeratePa		(* DerateLookUp *),		
				BatPNomMinPa_S	:=	BatPNomMinPa_S		(* REAL *),		
				BatPNomMaxPa_S	:=	BatPNomMaxPa_S		(* REAL *),		
				BatUMaxPa_S	:=	BatUMaxPa_S		(* REAL *),		
				BatUMinPa_S	:=	BatUMinPa_S		(* REAL *),
				Sys_Parameters	:=	Sys_Parameters	,
				BattTotalRackCntPa_S	:=	BattTotalRackCntPa_S(* USINT *),
				BattPartMinRackCntPa_S	:=	BattPartMinRackCntPa_S(* USINT *)
								
);										
PS[1].BMS.In.Param	:=	Ps_Sim_Param_2.BMS_Param_In;				
PS[1].Gc.In.Param	:=	Ps_Sim_Param_2.Gc_Param_In;
(*___________________________________________________________*)
(*Line Up 2*)
								
Ps_Sim_Param_2(										
				Gc_PQ_FU_RefSelPa_S	:=	Gc_PQ_FU_RefSelPa_S		(* INT *),			
				Gc_SNomPa_S	:=	Gc_SNomPa_S		(* REAL *),		
				Gc_fDroopPa_S	:=	Gc_fDroopPa_S		(* REAL *),		
				Gc_UDroopPa_S	:=	Gc_UDroopPa_S		(* REAL *),		
				Gc_TMotorPa_S	:=	Gc_TMotorPa_S		(* TIME *),		
				Gc_TExciterPa_S	:=	Gc_TExciterPa_S		(* TIME *),		
				Gc_P_UpPa_S	:=	Gc_P_UpPa_S		(* REAL *),		
				Gc_P_DownPa_S	:=	Gc_P_DownPa_S		(* REAL *),		
				Gc_PLimMinPa_S	:=	Gc_PLimMinPa_S		(* REAL *),		
				Gc_PLimMaxPa_S	:=	Gc_PLimMaxPa_S		(* REAL *),		
				Gc_PinitPa_S	:=	Gc_PinitPa_S		(* REAL *),		
				Gc_PNomPa_S	:=	Gc_PNomPa_S		(* REAL *),		
				Gc_QLimMinPa_S	:=	Gc_QLimMinPa_S		(* REAL *),		
				Gc_QLimMaxPa_S	:=	Gc_QLimMaxPa_S		(* REAL *),		
				Gc_QinitPa_S	:=	Gc_QinitPa_S		(* REAL *),		
				Gc_QNomPa_S	:=	Gc_QNomPa_S		(* REAL *),		
				Gc_OvPFactorPa_S	:=	Gc_OvPFactorPa_S		(* REAL *),		
				Gc_OvPLockInTPa_S	:=	Gc_OvPLockInTPa_S		(* TIME *),		
				Gc_OvQFactorPa_S	:=	Gc_OvQFactorPa_S		(* REAL *),		
				Gc_OvQLockInTPa_S	:=	Gc_OvQLockInTPa_S		(* TIME *),		
				Gc_OvUFactorPa_S	:=	Gc_OvUFactorPa_S		(* REAL *),		
				Gc_OvULockInTPa_S	:=	Gc_OvULockInTPa_S		(* TIME *),		
				Gc_OvFFactorPa_S	:=	Gc_OvFFactorPa_S		(* REAL *),		
				Gc_OvFLockInTPa_S	:=	Gc_OvFLockInTPa_S		(* TIME *),		
				BatUNomPa_S	:=	BatUNomPa_S		(* REAL *),		
				BatSNomPa_S	:=	BatSNomPa_S		(* REAL *),		
				BatEInitPa_S	:=	BatEInitPa_S		(* REAL *),		
				BatENomPa_S	:=	BatENomPa_S		(* REAL *),		
				BatEnDerateWrtSocPa_S	:=	BatEnDerateWrtSocPa_S		(* BOOL *),		
				BatEnDerateWrtTempPa_S	:=	BatEnDerateWrtTempPa_S		(* BOOL *),		
				BatDrtChrgOnSocLookUpSocPa	:=	BatDrtChrgOnSocLookUpSocPa		(* DerateLookUp *),		
				BatDrtChrgOnSocLookUpDrtPa	:=	BatDrtChrgOnSocLookUpDrtPa		(* DerateLookUp *),		
				BatDrtDChrgOnSocLookUpSocPa	:=	BatDrtDChrgOnSocLookUpSocPa		(* DerateLookUp *),		
				BatDrtDChrgOnSocLookUpDrtPa	:=	BatDrtDChrgOnSocLookUpDrtPa		(* DerateLookUp *),		
				BatDerateTempLookUpTempPa	:=	BatDerateTempLookUpTempPa		(* DerateLookUp *),		
				BatDerateTempLookUpDeratePa	:=	BatDerateTempLookUpDeratePa		(* DerateLookUp *),		
				BatPNomMinPa_S	:=	BatPNomMinPa_S		(* REAL *),		
				BatPNomMaxPa_S	:=	BatPNomMaxPa_S		(* REAL *),		
				BatUMaxPa_S	:=	BatUMaxPa_S		(* REAL *),		
				BatUMinPa_S	:=	BatUMinPa_S		(* REAL *),
				Sys_Parameters	:=	Sys_Parameters	,
				BattTotalRackCntPa_S	:=	BattTotalRackCntPa_S(* USINT *),
				BattPartMinRackCntPa_S	:=	BattPartMinRackCntPa_S(* USINT *)
								
);										
								
PS[2].BMS.In.Param	:=	Ps_Sim_Param_2.BMS_Param_In;				
PS[2].Gc.In.Param	:=	Ps_Sim_Param_2.Gc_Param_In;
(*___________________________________________________________*)
(*Line Up 3*)
								
Ps_Sim_Param_3(										
				Gc_PQ_FU_RefSelPa_S	:=	Gc_PQ_FU_RefSelPa_S		(* INT *),			
				Gc_SNomPa_S	:=	Gc_SNomPa_S		(* REAL *),		
				Gc_fDroopPa_S	:=	Gc_fDroopPa_S		(* REAL *),		
				Gc_UDroopPa_S	:=	Gc_UDroopPa_S		(* REAL *),		
				Gc_TMotorPa_S	:=	Gc_TMotorPa_S		(* TIME *),		
				Gc_TExciterPa_S	:=	Gc_TExciterPa_S		(* TIME *),		
				Gc_P_UpPa_S	:=	Gc_P_UpPa_S		(* REAL *),		
				Gc_P_DownPa_S	:=	Gc_P_DownPa_S		(* REAL *),		
				Gc_PLimMinPa_S	:=	Gc_PLimMinPa_S		(* REAL *),		
				Gc_PLimMaxPa_S	:=	Gc_PLimMaxPa_S		(* REAL *),		
				Gc_PinitPa_S	:=	Gc_PinitPa_S		(* REAL *),		
				Gc_PNomPa_S	:=	Gc_PNomPa_S		(* REAL *),		
				Gc_QLimMinPa_S	:=	Gc_QLimMinPa_S		(* REAL *),		
				Gc_QLimMaxPa_S	:=	Gc_QLimMaxPa_S		(* REAL *),		
				Gc_QinitPa_S	:=	Gc_QinitPa_S		(* REAL *),		
				Gc_QNomPa_S	:=	Gc_QNomPa_S		(* REAL *),		
				Gc_OvPFactorPa_S	:=	Gc_OvPFactorPa_S		(* REAL *),		
				Gc_OvPLockInTPa_S	:=	Gc_OvPLockInTPa_S		(* TIME *),		
				Gc_OvQFactorPa_S	:=	Gc_OvQFactorPa_S		(* REAL *),		
				Gc_OvQLockInTPa_S	:=	Gc_OvQLockInTPa_S		(* TIME *),		
				Gc_OvUFactorPa_S	:=	Gc_OvUFactorPa_S		(* REAL *),		
				Gc_OvULockInTPa_S	:=	Gc_OvULockInTPa_S		(* TIME *),		
				Gc_OvFFactorPa_S	:=	Gc_OvFFactorPa_S		(* REAL *),		
				Gc_OvFLockInTPa_S	:=	Gc_OvFLockInTPa_S		(* TIME *),		
				BatUNomPa_S	:=	BatUNomPa_S		(* REAL *),		
				BatSNomPa_S	:=	BatSNomPa_S		(* REAL *),		
				BatEInitPa_S	:=	BatEInitPa_S		(* REAL *),		
				BatENomPa_S	:=	BatENomPa_S		(* REAL *),		
				BatEnDerateWrtSocPa_S	:=	BatEnDerateWrtSocPa_S		(* BOOL *),		
				BatEnDerateWrtTempPa_S	:=	BatEnDerateWrtTempPa_S		(* BOOL *),		
				BatDrtChrgOnSocLookUpSocPa	:=	BatDrtChrgOnSocLookUpSocPa		(* DerateLookUp *),		
				BatDrtChrgOnSocLookUpDrtPa	:=	BatDrtChrgOnSocLookUpDrtPa		(* DerateLookUp *),		
				BatDrtDChrgOnSocLookUpSocPa	:=	BatDrtDChrgOnSocLookUpSocPa		(* DerateLookUp *),		
				BatDrtDChrgOnSocLookUpDrtPa	:=	BatDrtDChrgOnSocLookUpDrtPa		(* DerateLookUp *),		
				BatDerateTempLookUpTempPa	:=	BatDerateTempLookUpTempPa		(* DerateLookUp *),		
				BatDerateTempLookUpDeratePa	:=	BatDerateTempLookUpDeratePa		(* DerateLookUp *),		
				BatPNomMinPa_S	:=	BatPNomMinPa_S		(* REAL *),		
				BatPNomMaxPa_S	:=	BatPNomMaxPa_S		(* REAL *),		
				BatUMaxPa_S	:=	BatUMaxPa_S		(* REAL *),		
				BatUMinPa_S	:=	BatUMinPa_S		(* REAL *),
				Sys_Parameters	:=	Sys_Parameters	,
				BattTotalRackCntPa_S	:=	BattTotalRackCntPa_S(* USINT *),
				BattPartMinRackCntPa_S	:=	BattPartMinRackCntPa_S(* USINT *)
								
);										
PS[3].BMS.In.Param	:=	Ps_Sim_Param_3.BMS_Param_In;				
PS[3].Gc.In.Param	:=	Ps_Sim_Param_3.Gc_Param_In;
(*___________________________________________________________*)
(*Line Up 4*)
								
Ps_Sim_Param_4(										
				Gc_PQ_FU_RefSelPa_S	:=	Gc_PQ_FU_RefSelPa_S		(* INT *),			
				Gc_SNomPa_S	:=	Gc_SNomPa_S		(* REAL *),		
				Gc_fDroopPa_S	:=	Gc_fDroopPa_S		(* REAL *),		
				Gc_UDroopPa_S	:=	Gc_UDroopPa_S		(* REAL *),		
				Gc_TMotorPa_S	:=	Gc_TMotorPa_S		(* TIME *),		
				Gc_TExciterPa_S	:=	Gc_TExciterPa_S		(* TIME *),		
				Gc_P_UpPa_S	:=	Gc_P_UpPa_S		(* REAL *),		
				Gc_P_DownPa_S	:=	Gc_P_DownPa_S		(* REAL *),		
				Gc_PLimMinPa_S	:=	Gc_PLimMinPa_S		(* REAL *),		
				Gc_PLimMaxPa_S	:=	Gc_PLimMaxPa_S		(* REAL *),		
				Gc_PinitPa_S	:=	Gc_PinitPa_S		(* REAL *),		
				Gc_PNomPa_S	:=	Gc_PNomPa_S		(* REAL *),		
				Gc_QLimMinPa_S	:=	Gc_QLimMinPa_S		(* REAL *),		
				Gc_QLimMaxPa_S	:=	Gc_QLimMaxPa_S		(* REAL *),		
				Gc_QinitPa_S	:=	Gc_QinitPa_S		(* REAL *),		
				Gc_QNomPa_S	:=	Gc_QNomPa_S		(* REAL *),		
				Gc_OvPFactorPa_S	:=	Gc_OvPFactorPa_S		(* REAL *),		
				Gc_OvPLockInTPa_S	:=	Gc_OvPLockInTPa_S		(* TIME *),		
				Gc_OvQFactorPa_S	:=	Gc_OvQFactorPa_S		(* REAL *),		
				Gc_OvQLockInTPa_S	:=	Gc_OvQLockInTPa_S		(* TIME *),		
				Gc_OvUFactorPa_S	:=	Gc_OvUFactorPa_S		(* REAL *),		
				Gc_OvULockInTPa_S	:=	Gc_OvULockInTPa_S		(* TIME *),		
				Gc_OvFFactorPa_S	:=	Gc_OvFFactorPa_S		(* REAL *),		
				Gc_OvFLockInTPa_S	:=	Gc_OvFLockInTPa_S		(* TIME *),		
				BatUNomPa_S	:=	BatUNomPa_S		(* REAL *),		
				BatSNomPa_S	:=	BatSNomPa_S		(* REAL *),		
				BatEInitPa_S	:=	BatEInitPa_S		(* REAL *),		
				BatENomPa_S	:=	BatENomPa_S		(* REAL *),		
				BatEnDerateWrtSocPa_S	:=	BatEnDerateWrtSocPa_S		(* BOOL *),		
				BatEnDerateWrtTempPa_S	:=	BatEnDerateWrtTempPa_S		(* BOOL *),		
				BatDrtChrgOnSocLookUpSocPa	:=	BatDrtChrgOnSocLookUpSocPa		(* DerateLookUp *),		
				BatDrtChrgOnSocLookUpDrtPa	:=	BatDrtChrgOnSocLookUpDrtPa		(* DerateLookUp *),		
				BatDrtDChrgOnSocLookUpSocPa	:=	BatDrtDChrgOnSocLookUpSocPa		(* DerateLookUp *),		
				BatDrtDChrgOnSocLookUpDrtPa	:=	BatDrtDChrgOnSocLookUpDrtPa		(* DerateLookUp *),		
				BatDerateTempLookUpTempPa	:=	BatDerateTempLookUpTempPa		(* DerateLookUp *),		
				BatDerateTempLookUpDeratePa	:=	BatDerateTempLookUpDeratePa		(* DerateLookUp *),		
				BatPNomMinPa_S	:=	BatPNomMinPa_S		(* REAL *),		
				BatPNomMaxPa_S	:=	BatPNomMaxPa_S		(* REAL *),		
				BatUMaxPa_S	:=	BatUMaxPa_S		(* REAL *),		
				BatUMinPa_S	:=	BatUMinPa_S		(* REAL *),
				Sys_Parameters	:=	Sys_Parameters	,
				BattTotalRackCntPa_S	:=	BattTotalRackCntPa_S(* USINT *),
				BattPartMinRackCntPa_S	:=	BattPartMinRackCntPa_S(* USINT *)
								
);										
PS[4].BMS.In.Param	:=	Ps_Sim_Param_4.BMS_Param_In;				
PS[4].Gc.In.Param	:=	Ps_Sim_Param_4.Gc_Param_In;
(*___________________________________________________________*)
(*Line Up 5*)
Ps_Sim_Param_5(										
				Gc_PQ_FU_RefSelPa_S	:=	Gc_PQ_FU_RefSelPa_S		(* INT *),			
				Gc_SNomPa_S	:=	Gc_SNomPa_S		(* REAL *),		
				Gc_fDroopPa_S	:=	Gc_fDroopPa_S		(* REAL *),		
				Gc_UDroopPa_S	:=	Gc_UDroopPa_S		(* REAL *),		
				Gc_TMotorPa_S	:=	Gc_TMotorPa_S		(* TIME *),		
				Gc_TExciterPa_S	:=	Gc_TExciterPa_S		(* TIME *),		
				Gc_P_UpPa_S	:=	Gc_P_UpPa_S		(* REAL *),		
				Gc_P_DownPa_S	:=	Gc_P_DownPa_S		(* REAL *),		
				Gc_PLimMinPa_S	:=	Gc_PLimMinPa_S		(* REAL *),		
				Gc_PLimMaxPa_S	:=	Gc_PLimMaxPa_S		(* REAL *),		
				Gc_PinitPa_S	:=	Gc_PinitPa_S		(* REAL *),		
				Gc_PNomPa_S	:=	Gc_PNomPa_S		(* REAL *),		
				Gc_QLimMinPa_S	:=	Gc_QLimMinPa_S		(* REAL *),		
				Gc_QLimMaxPa_S	:=	Gc_QLimMaxPa_S		(* REAL *),		
				Gc_QinitPa_S	:=	Gc_QinitPa_S		(* REAL *),		
				Gc_QNomPa_S	:=	Gc_QNomPa_S		(* REAL *),		
				Gc_OvPFactorPa_S	:=	Gc_OvPFactorPa_S		(* REAL *),		
				Gc_OvPLockInTPa_S	:=	Gc_OvPLockInTPa_S		(* TIME *),		
				Gc_OvQFactorPa_S	:=	Gc_OvQFactorPa_S		(* REAL *),		
				Gc_OvQLockInTPa_S	:=	Gc_OvQLockInTPa_S		(* TIME *),		
				Gc_OvUFactorPa_S	:=	Gc_OvUFactorPa_S		(* REAL *),		
				Gc_OvULockInTPa_S	:=	Gc_OvULockInTPa_S		(* TIME *),		
				Gc_OvFFactorPa_S	:=	Gc_OvFFactorPa_S		(* REAL *),		
				Gc_OvFLockInTPa_S	:=	Gc_OvFLockInTPa_S		(* TIME *),		
				BatUNomPa_S	:=	BatUNomPa_S		(* REAL *),		
				BatSNomPa_S	:=	BatSNomPa_S		(* REAL *),		
				BatEInitPa_S	:=	BatEInitPa_S		(* REAL *),		
				BatENomPa_S	:=	BatENomPa_S		(* REAL *),		
				BatEnDerateWrtSocPa_S	:=	BatEnDerateWrtSocPa_S		(* BOOL *),		
				BatEnDerateWrtTempPa_S	:=	BatEnDerateWrtTempPa_S		(* BOOL *),		
				BatDrtChrgOnSocLookUpSocPa	:=	BatDrtChrgOnSocLookUpSocPa		(* DerateLookUp *),		
				BatDrtChrgOnSocLookUpDrtPa	:=	BatDrtChrgOnSocLookUpDrtPa		(* DerateLookUp *),		
				BatDrtDChrgOnSocLookUpSocPa	:=	BatDrtDChrgOnSocLookUpSocPa		(* DerateLookUp *),		
				BatDrtDChrgOnSocLookUpDrtPa	:=	BatDrtDChrgOnSocLookUpDrtPa		(* DerateLookUp *),		
				BatDerateTempLookUpTempPa	:=	BatDerateTempLookUpTempPa		(* DerateLookUp *),		
				BatDerateTempLookUpDeratePa	:=	BatDerateTempLookUpDeratePa		(* DerateLookUp *),		
				BatPNomMinPa_S	:=	BatPNomMinPa_S		(* REAL *),		
				BatPNomMaxPa_S	:=	BatPNomMaxPa_S		(* REAL *),		
				BatUMaxPa_S	:=	BatUMaxPa_S		(* REAL *),		
				BatUMinPa_S	:=	BatUMinPa_S		(* REAL *),
				Sys_Parameters	:=	Sys_Parameters	,
				BattTotalRackCntPa_S	:=	BattTotalRackCntPa_S(* USINT *),
				BattPartMinRackCntPa_S	:=	BattPartMinRackCntPa_S(* USINT *)
								
);										
PS[5].BMS.In.Param	:=	Ps_Sim_Param_5.BMS_Param_In;				
PS[5].Gc.In.Param	:=	Ps_Sim_Param_5.Gc_Param_In;
							
							(* Line 1 GC Modbus In*)
PSModbus_In_1(TDC_Cmd_In:=L1_Gc_Cmd_In_I);
L1_Gc_Cmd_In_Q:=PSModbus_In_1.TDC_Cmd_Out;
L1_Gc_Cmd_Rsp_Q:=PSModbus_In_1.TDC_Mon_Out;
PS[1].Gc.In.LuC :=PSModbus_In_1.Gc_LuC_In;
								
(*Line 1 BMS Modbus In	*)
BMSModbus_In_1(Cmd_IN	:=	L1_BMS_Cmd_In_I	);
L1_BMS_Cmd_In_Q		:=	BMSModbus_In_1.Cmd_FdBk;
L1_BMS_Cmd_Rsp_Q		:=	BMSModbus_In_1.Resp;
PS[1].BMS.In.LuC	:=	BMSModbus_In_1.BMS_Luc_IN;
(*___________________________________________________*)
(* Line 2 GC Modbus In*)
PSModbus_In_2(TDC_Cmd_In:=L2_Gc_Cmd_In_I);
L2_Gc_Cmd_In_Q:=PSModbus_In_2.TDC_Cmd_Out;
L2_Gc_Cmd_Rsp_Q:=PSModbus_In_2.TDC_Mon_Out;
PS[2].Gc.In.LuC :=PSModbus_In_2.Gc_LuC_In;
								
(*Line 2 BMS Modbus In	*)
BMSModbus_In_2(Cmd_IN	:=	L2_BMS_Cmd_In_I	);
L2_BMS_Cmd_In_Q		:=	BMSModbus_In_2.Cmd_FdBk;
L2_BMS_Cmd_Rsp_Q		:=	BMSModbus_In_2.Resp;
PS[2].BMS.In.LuC	:=	BMSModbus_In_2.BMS_Luc_IN;
(*___________________________________________________*)
(* Line 3 GC Modbus In*)
PSModbus_In_3(TDC_Cmd_In:=L3_Gc_Cmd_In_I);
L3_Gc_Cmd_In_Q:=PSModbus_In_3.TDC_Cmd_Out;
L3_Gc_Cmd_Rsp_Q:=PSModbus_In_3.TDC_Mon_Out;
PS[3].Gc.In.LuC :=PSModbus_In_3.Gc_LuC_In;
								
(*Line 3 BMS Modbus In	*)
BMSModbus_In_3(Cmd_IN	:=	L3_BMS_Cmd_In_I	);
L3_BMS_Cmd_In_Q		:=	BMSModbus_In_3.Cmd_FdBk;
L3_BMS_Cmd_Rsp_Q		:=	BMSModbus_In_3.Resp;
PS[3].BMS.In.LuC	:=	BMSModbus_In_3.BMS_Luc_IN;
(*___________________________________________________*)
(* Line 4 GC Modbus In*)
PSModbus_In_4(TDC_Cmd_In:=L4_Gc_Cmd_In_I);
L4_Gc_Cmd_In_Q:=PSModbus_In_4.TDC_Cmd_Out;
L4_Gc_Cmd_Rsp_Q:=PSModbus_In_4.TDC_Mon_Out;
PS[4].Gc.In.LuC :=PSModbus_In_4.Gc_LuC_In;
								
(*Line 4 BMS Modbus In	*)
BMSModbus_In_4(Cmd_IN	:=	L4_BMS_Cmd_In_I	);
L4_BMS_Cmd_In_Q		:=	BMSModbus_In_4.Cmd_FdBk;
L4_BMS_Cmd_Rsp_Q		:=	BMSModbus_In_4.Resp;
PS[4].BMS.In.LuC	:=	BMSModbus_In_4.BMS_Luc_IN;
(*___________________________________________________*)
(* Line 5 GC Modbus In*)
PSModbus_In_5(TDC_Cmd_In:=L5_Gc_Cmd_In_I);
L5_Gc_Cmd_In_Q:=PSModbus_In_5.TDC_Cmd_Out;
L5_Gc_Cmd_Rsp_Q:=PSModbus_In_5.TDC_Mon_Out;
PS[5].Gc.In.LuC :=PSModbus_In_5.Gc_LuC_In;
								
(*Line 5 BMS Modbus In	*)
BMSModbus_In_5(Cmd_IN	:=	L5_BMS_Cmd_In_I	);
L5_BMS_Cmd_In_Q		:=	BMSModbus_In_5.Cmd_FdBk;
L5_BMS_Cmd_Rsp_Q		:=	BMSModbus_In_5.Resp;
PS[5].BMS.In.LuC	:=	BMSModbus_In_5.BMS_Luc_IN;
								
(*___________________________________________________*)
Grid_Modbus_In_1(								
					Grid_01_CloseCmd_I	:=	Grid_01_CloseCmd_I	,
					Grid_01_OpenCmd_I	:=	Grid_01_OpenCmd_I	,
					Grid_01_AlarmReset_I	:=	Grid_01_AlarmReset_I	
					);			
Grid_01_AlarmReset_Q	:=	Grid_Modbus_In_1.Grid_01_AlarmReset_Q;						
Grid_01_OpenCmd_Q	:=	Grid_Modbus_In_1.Grid_01_OpenCmd_Q;						
Grid_01_CloseCmd_Q	:=	Grid_Modbus_In_1.Grid_01_CloseCmd_Q;						
Grid_Dat[1].Grid_In	:=	Grid_Modbus_In_1.Grid_In;						
								
								
								
								
Fed_ModInBlock_1(								
					Fed_01_AlarmReset_I	:=	Fed_01_AlarmReset_I	,
					Fed_01_OpenCmd_I	:=	Fed_01_OpenCmd_I	,
					Fed_01_CloseCmd_I	:=	Fed_01_CloseCmd_I	
					);			
Fed_Data[1].Fed_ModBus_In	:=	Fed_ModInBlock_1.Fed_ModBus_In	;					
Fed_01_CloseCmd_Q	:=	Fed_ModInBlock_1.Fed_01_CloseCmd_Q	;					
Fed_01_OpenCmd_Q	:=	Fed_ModInBlock_1.Fed_01_OpenCmd_Q	;					
Fed_01_AlarmReset_Q	:=	Fed_ModInBlock_1.Fed_01_AlarmReset_Q	;
							
							Grid_Var_In_1();
Grid_Dat[1].Grid_HMI_In  	:=	Grid_Var_In_1.Grid_HMI_In;
								
Grid_HMI_Var_In_1();
								
								
Fed_Var_In_1();
Fed_Data[1].Feeder_In		:=	Fed_Var_In_1.Feeder_Var_IN;
								
PS_Var_In_1(							
				GcStartCmd_S		:=	PS1_GcStartCmd_S	,
				GcStopCmd_S			:=	PS1_GcStopCmd_S	,
				GcBreakerCloseCmd_S	:=	PS1_GcBreakerCloseCmd_S	,
				GcBreakerOpenCmd_S	:=	PS1_GcBreakerOpenCmd_S	,
				GcAlarmReset_S		:=	PS1_GcBreakerOpenCmd_S	,
				GcSim_CritAl_S		:=	PS1_GcSim_CritAl_S	,
				GcSim_NonCritAl_S	:=	PS1_GcSim_NonCritAl_S	,
				GcSim_WarnAl_S		:=	PS1_GcSim_WarnAl_S	,
				GcEStop_S			:=	PS1_GcEStop_S	,
				BattStartCmd_S		:=	PS1_BattStartCmd_S	,
				BattStopCmd_S		:=	PS1_BattStopCmd_S	,
				BattAlarmReset_S	:=	PS1_BattAlarmReset_S	,
				BattSim_CritAl_S	:=	PS1_BattSim_CritAl_S	,
				BattSim_NonCritAl_S	:=	PS1_BattSim_NonCritAl_S	,
				BattSim_WarnAl_S	:=	PS1_BattSim_WarnAl_S	,
				BattEStop_S			:=	PS1_BattEStop_S	,
				BattSim_FireAl_S	:=	PS1_BattSim_FireAl_S	,
				Rk1InService_S		:=	PS1_Rk1InService_S	,
				Rk1RkCloseCmd_S		:=	PS1_Rk1RkCloseCmd_S	,
				Rk1RkOpenCmd_S		:=	PS1_Rk1RkOpenCmd_S	,
				Rk1RkAlarm_S		:=	PS1_Rk1RkAlarm_S	,
				Rk2InService_S		:=	PS1_Rk2InService_S	,
				Rk2RkCloseCmd_S		:=	PS1_Rk2RkCloseCmd_S	,
				Rk2RkOpenCmd_S		:=	PS1_Rk2RkOpenCmd_S	,
				Rk2RkAlarm_S		:=	PS1_Rk2RkAlarm_S	,
				Rk3InService_S		:=	PS1_Rk3InService_S	,
				Rk3RkCloseCmd_S		:=	PS1_Rk3RkCloseCmd_S	,
				Rk3RkOpenCmd_S		:=	PS1_Rk3RkOpenCmd_S	,
				Rk3RkAlarm_S		:=	PS1_Rk3RkAlarm_S	,
				Rk4InService_S		:=	PS1_Rk4InService_S	,
				Rk4RkCloseCmd_S		:=	PS1_Rk4RkCloseCmd_S	,
				Rk4RkOpenCmd_S		:=	PS1_Rk4RkOpenCmd_S	,
				Rk4RkAlarm_S		:=	PS1_Rk4RkAlarm_S	,
				Rk5InService_S		:=	PS1_Rk5InService_S	,
				Rk5RkCloseCmd_S		:=	PS1_Rk5RkCloseCmd_S	,
				Rk5RkOpenCmd_S		:=	PS1_Rk5RkOpenCmd_S	,
				Rk5RkAlarm_S		:=	PS1_Rk5RkAlarm_S	
							
				);			
								
PS[1].Gc.In.HMI 	:=	PS_Var_In_1.Gc_HMI_In;
PS[1].BMS.In.HMI	:=	PS_Var_In_1.BMS_HMI_In;
								
PS_Var_In_2(							
				GcStartCmd_S		:=	PS1_GcStartCmd_S	,
				GcStopCmd_S			:=	PS1_GcStopCmd_S	,
				GcBreakerCloseCmd_S	:=	PS1_GcBreakerCloseCmd_S	,
				GcBreakerOpenCmd_S	:=	PS1_GcBreakerOpenCmd_S	,
				GcAlarmReset_S		:=	PS1_GcBreakerOpenCmd_S	,
				GcSim_CritAl_S		:=	PS1_GcSim_CritAl_S	,
				GcSim_NonCritAl_S	:=	PS1_GcSim_NonCritAl_S	,
				GcSim_WarnAl_S		:=	PS1_GcSim_WarnAl_S	,
				GcEStop_S			:=	PS1_GcEStop_S	,
				BattStartCmd_S		:=	PS1_BattStartCmd_S	,
				BattStopCmd_S		:=	PS1_BattStopCmd_S	,
				BattAlarmReset_S	:=	PS1_BattAlarmReset_S	,
				BattSim_CritAl_S	:=	PS1_BattSim_CritAl_S	,
				BattSim_NonCritAl_S	:=	PS1_BattSim_NonCritAl_S	,
				BattSim_WarnAl_S	:=	PS1_BattSim_WarnAl_S	,
				BattEStop_S			:=	PS1_BattEStop_S	,
				BattSim_FireAl_S	:=	PS1_BattSim_FireAl_S	,
				Rk1InService_S		:=	PS1_Rk1InService_S	,
				Rk1RkCloseCmd_S		:=	PS1_Rk1RkCloseCmd_S	,
				Rk1RkOpenCmd_S		:=	PS1_Rk1RkOpenCmd_S	,
				Rk1RkAlarm_S		:=	PS1_Rk1RkAlarm_S	,
				Rk2InService_S		:=	PS1_Rk2InService_S	,
				Rk2RkCloseCmd_S		:=	PS1_Rk2RkCloseCmd_S	,
				Rk2RkOpenCmd_S		:=	PS1_Rk2RkOpenCmd_S	,
				Rk2RkAlarm_S		:=	PS1_Rk2RkAlarm_S	,
				Rk3InService_S		:=	PS1_Rk3InService_S	,
				Rk3RkCloseCmd_S		:=	PS1_Rk3RkCloseCmd_S	,
				Rk3RkOpenCmd_S		:=	PS1_Rk3RkOpenCmd_S	,
				Rk3RkAlarm_S		:=	PS1_Rk3RkAlarm_S	,
				Rk4InService_S		:=	PS1_Rk4InService_S	,
				Rk4RkCloseCmd_S		:=	PS1_Rk4RkCloseCmd_S	,
				Rk4RkOpenCmd_S		:=	PS1_Rk4RkOpenCmd_S	,
				Rk4RkAlarm_S		:=	PS1_Rk4RkAlarm_S	,
				Rk5InService_S		:=	PS1_Rk5InService_S	,
				Rk5RkCloseCmd_S		:=	PS1_Rk5RkCloseCmd_S	,
				Rk5RkOpenCmd_S		:=	PS1_Rk5RkOpenCmd_S	,
				Rk5RkAlarm_S		:=	PS1_Rk5RkAlarm_S	
							
				);			
								
PS[2].Gc.In.HMI 	:=	PS_Var_In_2.Gc_HMI_In;
PS[2].BMS.In.HMI	:=	PS_Var_In_2.BMS_HMI_In;
								
PS_Var_In_3(							
				GcStartCmd_S		:=	PS1_GcStartCmd_S	,
				GcStopCmd_S			:=	PS1_GcStopCmd_S	,
				GcBreakerCloseCmd_S	:=	PS1_GcBreakerCloseCmd_S	,
				GcBreakerOpenCmd_S	:=	PS1_GcBreakerOpenCmd_S	,
				GcAlarmReset_S		:=	PS1_GcBreakerOpenCmd_S	,
				GcSim_CritAl_S		:=	PS1_GcSim_CritAl_S	,
				GcSim_NonCritAl_S	:=	PS1_GcSim_NonCritAl_S	,
				GcSim_WarnAl_S		:=	PS1_GcSim_WarnAl_S	,
				GcEStop_S			:=	PS1_GcEStop_S	,
				BattStartCmd_S		:=	PS1_BattStartCmd_S	,
				BattStopCmd_S		:=	PS1_BattStopCmd_S	,
				BattAlarmReset_S	:=	PS1_BattAlarmReset_S	,
				BattSim_CritAl_S	:=	PS1_BattSim_CritAl_S	,
				BattSim_NonCritAl_S	:=	PS1_BattSim_NonCritAl_S	,
				BattSim_WarnAl_S	:=	PS1_BattSim_WarnAl_S	,
				BattEStop_S			:=	PS1_BattEStop_S	,
				BattSim_FireAl_S	:=	PS1_BattSim_FireAl_S	,
				Rk1InService_S		:=	PS1_Rk1InService_S	,
				Rk1RkCloseCmd_S		:=	PS1_Rk1RkCloseCmd_S	,
				Rk1RkOpenCmd_S		:=	PS1_Rk1RkOpenCmd_S	,
				Rk1RkAlarm_S		:=	PS1_Rk1RkAlarm_S	,
				Rk2InService_S		:=	PS1_Rk2InService_S	,
				Rk2RkCloseCmd_S		:=	PS1_Rk2RkCloseCmd_S	,
				Rk2RkOpenCmd_S		:=	PS1_Rk2RkOpenCmd_S	,
				Rk2RkAlarm_S		:=	PS1_Rk2RkAlarm_S	,
				Rk3InService_S		:=	PS1_Rk3InService_S	,
				Rk3RkCloseCmd_S		:=	PS1_Rk3RkCloseCmd_S	,
				Rk3RkOpenCmd_S		:=	PS1_Rk3RkOpenCmd_S	,
				Rk3RkAlarm_S		:=	PS1_Rk3RkAlarm_S	,
				Rk4InService_S		:=	PS1_Rk4InService_S	,
				Rk4RkCloseCmd_S		:=	PS1_Rk4RkCloseCmd_S	,
				Rk4RkOpenCmd_S		:=	PS1_Rk4RkOpenCmd_S	,
				Rk4RkAlarm_S		:=	PS1_Rk4RkAlarm_S	,
				Rk5InService_S		:=	PS1_Rk5InService_S	,
				Rk5RkCloseCmd_S		:=	PS1_Rk5RkCloseCmd_S	,
				Rk5RkOpenCmd_S		:=	PS1_Rk5RkOpenCmd_S	,
				Rk5RkAlarm_S		:=	PS1_Rk5RkAlarm_S	
							
				);			
								
PS[3].Gc.In.HMI 	:=	PS_Var_In_3.Gc_HMI_In;
PS[3].BMS.In.HMI	:=	PS_Var_In_3.BMS_HMI_In;
								
PS_Var_In_4(							
				GcStartCmd_S		:=	PS1_GcStartCmd_S	,
				GcStopCmd_S			:=	PS1_GcStopCmd_S	,
				GcBreakerCloseCmd_S	:=	PS1_GcBreakerCloseCmd_S	,
				GcBreakerOpenCmd_S	:=	PS1_GcBreakerOpenCmd_S	,
				GcAlarmReset_S		:=	PS1_GcBreakerOpenCmd_S	,
				GcSim_CritAl_S		:=	PS1_GcSim_CritAl_S	,
				GcSim_NonCritAl_S	:=	PS1_GcSim_NonCritAl_S	,
				GcSim_WarnAl_S		:=	PS1_GcSim_WarnAl_S	,
				GcEStop_S			:=	PS1_GcEStop_S	,
				BattStartCmd_S		:=	PS1_BattStartCmd_S	,
				BattStopCmd_S		:=	PS1_BattStopCmd_S	,
				BattAlarmReset_S	:=	PS1_BattAlarmReset_S	,
				BattSim_CritAl_S	:=	PS1_BattSim_CritAl_S	,
				BattSim_NonCritAl_S	:=	PS1_BattSim_NonCritAl_S	,
				BattSim_WarnAl_S	:=	PS1_BattSim_WarnAl_S	,
				BattEStop_S			:=	PS1_BattEStop_S	,
				BattSim_FireAl_S	:=	PS1_BattSim_FireAl_S	,
				Rk1InService_S		:=	PS1_Rk1InService_S	,
				Rk1RkCloseCmd_S		:=	PS1_Rk1RkCloseCmd_S	,
				Rk1RkOpenCmd_S		:=	PS1_Rk1RkOpenCmd_S	,
				Rk1RkAlarm_S		:=	PS1_Rk1RkAlarm_S	,
				Rk2InService_S		:=	PS1_Rk2InService_S	,
				Rk2RkCloseCmd_S		:=	PS1_Rk2RkCloseCmd_S	,
				Rk2RkOpenCmd_S		:=	PS1_Rk2RkOpenCmd_S	,
				Rk2RkAlarm_S		:=	PS1_Rk2RkAlarm_S	,
				Rk3InService_S		:=	PS1_Rk3InService_S	,
				Rk3RkCloseCmd_S		:=	PS1_Rk3RkCloseCmd_S	,
				Rk3RkOpenCmd_S		:=	PS1_Rk3RkOpenCmd_S	,
				Rk3RkAlarm_S		:=	PS1_Rk3RkAlarm_S	,
				Rk4InService_S		:=	PS1_Rk4InService_S	,
				Rk4RkCloseCmd_S		:=	PS1_Rk4RkCloseCmd_S	,
				Rk4RkOpenCmd_S		:=	PS1_Rk4RkOpenCmd_S	,
				Rk4RkAlarm_S		:=	PS1_Rk4RkAlarm_S	,
				Rk5InService_S		:=	PS1_Rk5InService_S	,
				Rk5RkCloseCmd_S		:=	PS1_Rk5RkCloseCmd_S	,
				Rk5RkOpenCmd_S		:=	PS1_Rk5RkOpenCmd_S	,
				Rk5RkAlarm_S		:=	PS1_Rk5RkAlarm_S	
							
				);			
								
PS[4].Gc.In.HMI 	:=	PS_Var_In_4.Gc_HMI_In;
PS[4].BMS.In.HMI	:=	PS_Var_In_4.BMS_HMI_In;
								
PS_Var_In_5(							
				GcStartCmd_S		:=	PS1_GcStartCmd_S	,
				GcStopCmd_S			:=	PS1_GcStopCmd_S	,
				GcBreakerCloseCmd_S	:=	PS1_GcBreakerCloseCmd_S	,
				GcBreakerOpenCmd_S	:=	PS1_GcBreakerOpenCmd_S	,
				GcAlarmReset_S		:=	PS1_GcBreakerOpenCmd_S	,
				GcSim_CritAl_S		:=	PS1_GcSim_CritAl_S	,
				GcSim_NonCritAl_S	:=	PS1_GcSim_NonCritAl_S	,
				GcSim_WarnAl_S		:=	PS1_GcSim_WarnAl_S	,
				GcEStop_S			:=	PS1_GcEStop_S	,
				BattStartCmd_S		:=	PS1_BattStartCmd_S	,
				BattStopCmd_S		:=	PS1_BattStopCmd_S	,
				BattAlarmReset_S	:=	PS1_BattAlarmReset_S	,
				BattSim_CritAl_S	:=	PS1_BattSim_CritAl_S	,
				BattSim_NonCritAl_S	:=	PS1_BattSim_NonCritAl_S	,
				BattSim_WarnAl_S	:=	PS1_BattSim_WarnAl_S	,
				BattEStop_S			:=	PS1_BattEStop_S	,
				BattSim_FireAl_S	:=	PS1_BattSim_FireAl_S	,
				Rk1InService_S		:=	PS1_Rk1InService_S	,
				Rk1RkCloseCmd_S		:=	PS1_Rk1RkCloseCmd_S	,
				Rk1RkOpenCmd_S		:=	PS1_Rk1RkOpenCmd_S	,
				Rk1RkAlarm_S		:=	PS1_Rk1RkAlarm_S	,
				Rk2InService_S		:=	PS1_Rk2InService_S	,
				Rk2RkCloseCmd_S		:=	PS1_Rk2RkCloseCmd_S	,
				Rk2RkOpenCmd_S		:=	PS1_Rk2RkOpenCmd_S	,
				Rk2RkAlarm_S		:=	PS1_Rk2RkAlarm_S	,
				Rk3InService_S		:=	PS1_Rk3InService_S	,
				Rk3RkCloseCmd_S		:=	PS1_Rk3RkCloseCmd_S	,
				Rk3RkOpenCmd_S		:=	PS1_Rk3RkOpenCmd_S	,
				Rk3RkAlarm_S		:=	PS1_Rk3RkAlarm_S	,
				Rk4InService_S		:=	PS1_Rk4InService_S	,
				Rk4RkCloseCmd_S		:=	PS1_Rk4RkCloseCmd_S	,
				Rk4RkOpenCmd_S		:=	PS1_Rk4RkOpenCmd_S	,
				Rk4RkAlarm_S		:=	PS1_Rk4RkAlarm_S	,
				Rk5InService_S		:=	PS1_Rk5InService_S	,
				Rk5RkCloseCmd_S		:=	PS1_Rk5RkCloseCmd_S	,
				Rk5RkOpenCmd_S		:=	PS1_Rk5RkOpenCmd_S	,
				Rk5RkAlarm_S		:=	PS1_Rk5RkAlarm_S	
							
				);			
								
PS[5].Gc.In.HMI 	:=	PS_Var_In_5.Gc_HMI_In;
PS[5].BMS.In.HMI	:=	PS_Var_In_5.BMS_HMI_In;
							
						
					
END_PROGRAM

PROGRAM emCBSSim01_Ps01
  VAR
    Gc_1 : Gc;
    BMS_1 : BMS;
    Gc_2 : Gc;
    BMS_2 : BMS;
    Gc_3 : Gc;
    BMS_3 : BMS;
    Gc_4 : Gc;
    BMS_4 : BMS;
    Gc_5 : Gc;
    BMS_5 : BMS;
  END_VAR
  VAR_EXTERNAL
    PS : Ps_LineUP;
    PLC_TICKS_PER_SEC : INT;
    TStep : TIME;
    Sys_Data : Sys_Data;
  END_VAR
  VAR
    PLCCycle_1 : PLCCycle;
    Cpu_Fun_1 : Cpu_Fun;
  END_VAR

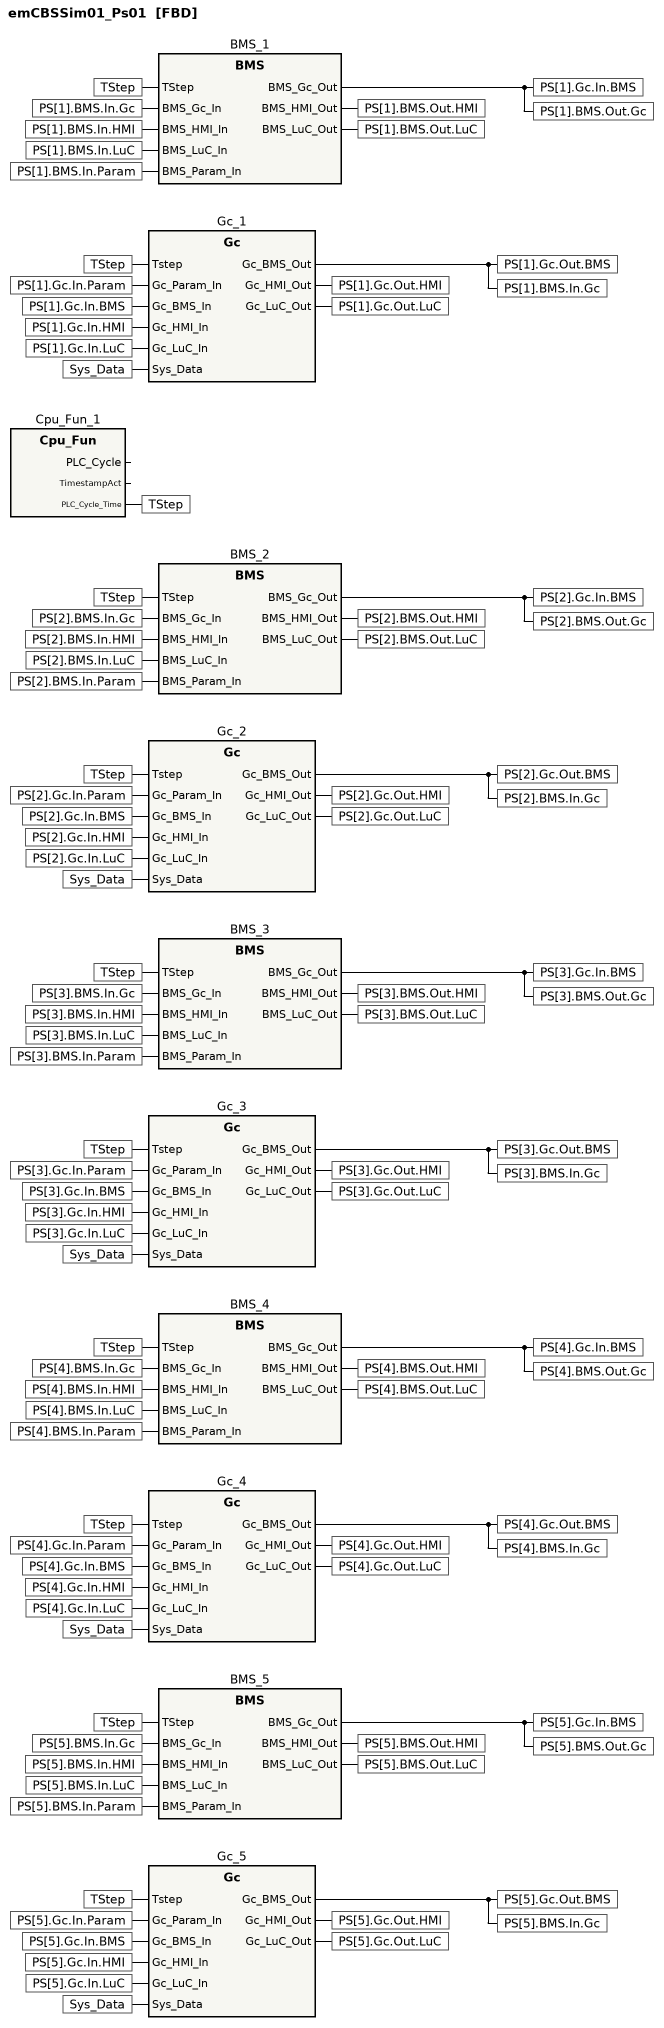
(* FBD diagram, written out as Structured Text *)
BMS_1(TStep := TStep, BMS_Gc_In := PS[1].BMS.In.Gc, BMS_HMI_In := PS[1].BMS.In.HMI, BMS_LuC_In := PS[1].BMS.In.LuC, BMS_Param_In := PS[1].BMS.In.Param);
PS[1].BMS.Out.HMI := BMS_1.BMS_HMI_Out;
PS[1].Gc.In.BMS := BMS_1.BMS_Gc_Out;
Gc_1(Tstep := TStep, Gc_Param_In := PS[1].Gc.In.Param, Gc_BMS_In := PS[1].Gc.In.BMS, Gc_HMI_In := PS[1].Gc.In.HMI, Gc_LuC_In := PS[1].Gc.In.LuC, Sys_Data := Sys_Data);
PS[1].BMS.In.Gc := Gc_1.Gc_BMS_Out;
Cpu_Fun_1();
TStep := Cpu_Fun_1.PLC_Cycle_Time;
PS[1].BMS.Out.LuC := BMS_1.BMS_LuC_Out;
PS[1].BMS.Out.Gc := BMS_1.BMS_Gc_Out;
PS[1].Gc.Out.HMI := Gc_1.Gc_HMI_Out;
PS[1].Gc.Out.LuC := Gc_1.Gc_LuC_Out;
PS[1].Gc.Out.BMS := Gc_1.Gc_BMS_Out;
BMS_2(TStep := TStep, BMS_Gc_In := PS[2].BMS.In.Gc, BMS_HMI_In := PS[2].BMS.In.HMI, BMS_LuC_In := PS[2].BMS.In.LuC, BMS_Param_In := PS[2].BMS.In.Param);
PS[2].BMS.Out.HMI := BMS_2.BMS_HMI_Out;
PS[2].Gc.In.BMS := BMS_2.BMS_Gc_Out;
Gc_2(Tstep := TStep, Gc_Param_In := PS[2].Gc.In.Param, Gc_BMS_In := PS[2].Gc.In.BMS, Gc_HMI_In := PS[2].Gc.In.HMI, Gc_LuC_In := PS[2].Gc.In.LuC, Sys_Data := Sys_Data);
PS[2].BMS.In.Gc := Gc_2.Gc_BMS_Out;
PS[2].BMS.Out.LuC := BMS_2.BMS_LuC_Out;
PS[2].BMS.Out.Gc := BMS_2.BMS_Gc_Out;
PS[2].Gc.Out.HMI := Gc_2.Gc_HMI_Out;
PS[2].Gc.Out.LuC := Gc_2.Gc_LuC_Out;
PS[2].Gc.Out.BMS := Gc_2.Gc_BMS_Out;
BMS_3(TStep := TStep, BMS_Gc_In := PS[3].BMS.In.Gc, BMS_HMI_In := PS[3].BMS.In.HMI, BMS_LuC_In := PS[3].BMS.In.LuC, BMS_Param_In := PS[3].BMS.In.Param);
PS[3].BMS.Out.HMI := BMS_3.BMS_HMI_Out;
PS[3].Gc.In.BMS := BMS_3.BMS_Gc_Out;
PS[3].BMS.Out.LuC := BMS_3.BMS_LuC_Out;
PS[3].BMS.Out.Gc := BMS_3.BMS_Gc_Out;
Gc_3(Tstep := TStep, Gc_Param_In := PS[3].Gc.In.Param, Gc_BMS_In := PS[3].Gc.In.BMS, Gc_HMI_In := PS[3].Gc.In.HMI, Gc_LuC_In := PS[3].Gc.In.LuC, Sys_Data := Sys_Data);
PS[3].Gc.Out.HMI := Gc_3.Gc_HMI_Out;
PS[3].Gc.Out.LuC := Gc_3.Gc_LuC_Out;
PS[3].Gc.Out.BMS := Gc_3.Gc_BMS_Out;
PS[3].BMS.In.Gc := Gc_3.Gc_BMS_Out;
BMS_4(TStep := TStep, BMS_Gc_In := PS[4].BMS.In.Gc, BMS_HMI_In := PS[4].BMS.In.HMI, BMS_LuC_In := PS[4].BMS.In.LuC, BMS_Param_In := PS[4].BMS.In.Param);
PS[4].BMS.Out.HMI := BMS_4.BMS_HMI_Out;
PS[4].Gc.In.BMS := BMS_4.BMS_Gc_Out;
Gc_4(Tstep := TStep, Gc_Param_In := PS[4].Gc.In.Param, Gc_BMS_In := PS[4].Gc.In.BMS, Gc_HMI_In := PS[4].Gc.In.HMI, Gc_LuC_In := PS[4].Gc.In.LuC, Sys_Data := Sys_Data);
PS[4].BMS.In.Gc := Gc_4.Gc_BMS_Out;
PS[4].BMS.Out.LuC := BMS_4.BMS_LuC_Out;
PS[4].BMS.Out.Gc := BMS_4.BMS_Gc_Out;
PS[4].Gc.Out.HMI := Gc_4.Gc_HMI_Out;
PS[4].Gc.Out.LuC := Gc_4.Gc_LuC_Out;
PS[4].Gc.Out.BMS := Gc_4.Gc_BMS_Out;
BMS_5(TStep := TStep, BMS_Gc_In := PS[5].BMS.In.Gc, BMS_HMI_In := PS[5].BMS.In.HMI, BMS_LuC_In := PS[5].BMS.In.LuC, BMS_Param_In := PS[5].BMS.In.Param);
PS[5].BMS.Out.HMI := BMS_5.BMS_HMI_Out;
PS[5].Gc.In.BMS := BMS_5.BMS_Gc_Out;
PS[5].BMS.Out.LuC := BMS_5.BMS_LuC_Out;
PS[5].BMS.Out.Gc := BMS_5.BMS_Gc_Out;
Gc_5(Tstep := TStep, Gc_Param_In := PS[5].Gc.In.Param, Gc_BMS_In := PS[5].Gc.In.BMS, Gc_HMI_In := PS[5].Gc.In.HMI, Gc_LuC_In := PS[5].Gc.In.LuC, Sys_Data := Sys_Data);
PS[5].Gc.Out.HMI := Gc_5.Gc_HMI_Out;
PS[5].Gc.Out.LuC := Gc_5.Gc_LuC_Out;
PS[5].Gc.Out.BMS := Gc_5.Gc_BMS_Out;
PS[5].BMS.In.Gc := Gc_5.Gc_BMS_Out;
END_PROGRAM

PROGRAM emCBSSim11_Out
  VAR
    BMSModbus_Out_1 : BMSModbus_Out;
    BMSModbus_Out_2 : BMSModbus_Out;
    BMSModbus_Out_3 : BMSModbus_Out;
    BMSModbus_Out_4 : BMSModbus_Out;
    BMSModbus_Out_5 : BMSModbus_Out;
  END_VAR
  VAR_EXTERNAL
    PS : Ps_LineUP;
  END_VAR
  VAR
    BMS_MB : BatSimMBData;
    BMS2_MB : BatSimMBData;
    BMS3_MB : BatSimMBData;
    BMS4_MB : BatSimMBData;
    BMS5_MB : BatSimMBData;
    BMS_Read_In_I : TDC;
    BMS_Read_In_Q : TDC;
    BMS_Read_Resp_Q : TDC;
    FedMod_Out_1 : FedMod_Out;
  END_VAR
  VAR_EXTERNAL
    Grid_Dat : Grid_Dat;
    Fed_Data : Feeder_Data;
  END_VAR
  VAR
    Fed_01_PAct_Q : MFI;
    Fed_01_EAct_Q : MFI;
    Fed_01_EExportAct_Q : MFI;
    Fed_01_EImportAct_Q : MFI;
    Fed_01_ExportKvarhAct_Q : MFI;
    Fed_01_FAct_Q : MFI;
    Fed_01_I1Act_Q : MFI;
    Fed_01_I2Act_Q : MFI;
    Fed_01_I3Act_Q : MFI;
    Fed_01_IAvgAct_Q : MFI;
    Fed_01_KvarhAct_Q : MFI;
    Fed_01_ImportKvarhAct_Q : MFI;
    Fed_01_Line_Q : MFI;
    Fed_01_PfAct_Q : MFI;
    Fed_01_QAct_Q : MFI;
    Fed_01_SAct_Q : MFI;
    Fed_01_U123AvgAct_Q : MFI;
    Fed_01_U12Act_Q : MFI;
    Fed_01_U1nAct_Q : MFI;
    Fed_01_U23Act_Q : MFI;
    Fed_01_U2nAct_Q : MFI;
    Fed_01_U31Act_Q : MFI;
    Fed_01_U3nAct_Q : MFI;
    Fed_01_UAct_Q : MFI;
    PSModbus_Out_1 : PSModbus_Out;
    PSModbus_Out_2 : PSModbus_Out;
    PSModbus_Out_3 : PSModbus_Out;
    PSModbus_Out_4 : PSModbus_Out;
    PSModbus_Out_5 : PSModbus_Out;
    TDC_Read_In : TDC;
    TDC_Read_Out : TDC;
    TDC_ReadData_Out : TDC;
    L1_Gc_Read_Rsp_Q : TDC;
    L1_Gc_Read_In_Q : TDC;
    L1_Gc_Read_In_I : TDC;
    L1_BMS_Read_In_Q : TDC;
    L1_BMS_Read_In_I : TDC;
    L1_BMS_Read_Resp_Q : TDC;
    L2_Gc_Read_Rsp_Q : TDC;
    L2_Gc_Read_In_Q : TDC;
    L2_Gc_Read_In_I : TDC;
    L2_BMS_Read_In_Q : TDC;
    L2_BMS_Read_In_I : TDC;
    L2_BMS_Read_Resp_Q : TDC;
    L3_Gc_Read_Rsp_Q : TDC;
    L3_Gc_Read_In_Q : TDC;
    L3_Gc_Read_In_I : TDC;
    L3_BMS_Read_In_Q : TDC;
    L3_BMS_Read_In_I : TDC;
    L3_BMS_Read_Resp_Q : TDC;
    L4_Gc_Read_Rsp_Q : TDC;
    L4_Gc_Read_In_Q : TDC;
    L4_Gc_Read_In_I : TDC;
    L4_BMS_Read_In_Q : TDC;
    L4_BMS_Read_In_I : TDC;
    L4_BMS_Read_Resp_Q : TDC;
    L5_Gc_Read_Rsp_Q : TDC;
    L5_Gc_Read_In_Q : TDC;
    L5_Gc_Read_In_I : TDC;
    L5_BMS_Read_In_Q : TDC;
    L5_BMS_Read_In_I : TDC;
    L5_BMS_Read_Resp_Q : TDC;
  END_VAR

						
							(* Line 1 GC Modbus Out*)
								
PSModbus_Out_1(	TDC_Read_In:=L1_Gc_Read_In_I(* TDC *),
				Gc_LuC_Out:= PS[1].Gc.Out.LuC (* Gc_LuC_Out *));
L1_Gc_Read_In_Q:=PSModbus_Out_1.TDC_Read_Out;
L1_Gc_Read_Rsp_Q:=PSModbus_Out_1.TDC_ReadData_Out;
								
(*Line 1 BMS Modbus Out	*)
BMSModbus_Out_1(
					TDC_cmd_I				:=		L1_BMS_Read_In_I ,
					BMS_Sys					:=		PS[1].BMS.Out.LuC.BatSimBMS_Sys,
					TotalRackNbPa			:=		PS[1].BMS.In.Param.TotalRackCntPa,
					BatSim_Rack_Array		:=		PS[1].BMS.Out.LuC.BatSim_Rack_Array
					)	;	
L1_BMS_Read_In_Q			:=	BMSModbus_Out_1.TDC_cmd_Q		;	
L1_BMS_Read_Resp_Q			:=	BMSModbus_Out_1.TDC_mon_Q		;	
BMS_MB 					:=	BMSModbus_Out_1.BMS_MD		;	
(*_______________________________________________*)
(* Line 2 GC Modbus Out*)
								
PSModbus_Out_2(	TDC_Read_In:=L2_Gc_Read_In_I(* TDC *),
				Gc_LuC_Out:= PS[2].Gc.Out.LuC (* Gc_LuC_Out *));
L2_Gc_Read_In_Q:=PSModbus_Out_2.TDC_Read_Out;
L2_Gc_Read_Rsp_Q:=PSModbus_Out_2.TDC_ReadData_Out;
								
(*Line 2 BMS Modbus Out	*)
BMSModbus_Out_2(
					TDC_cmd_I				:=		L2_BMS_Read_In_I ,
					BMS_Sys					:=		PS[2].BMS.Out.LuC.BatSimBMS_Sys,
					TotalRackNbPa			:=		PS[2].BMS.In.Param.TotalRackCntPa,
					BatSim_Rack_Array		:=		PS[2].BMS.Out.LuC.BatSim_Rack_Array
					)	;	
L2_BMS_Read_In_Q			:=	BMSModbus_Out_2.TDC_cmd_Q		;	
L2_BMS_Read_Resp_Q			:=	BMSModbus_Out_2.TDC_mon_Q		;	
BMS2_MB 					:=	BMSModbus_Out_2.BMS_MD		;	
								
(*_______________________________________________*)
(* Line 3 GC Modbus Out*)
								
PSModbus_Out_3(	TDC_Read_In:=L3_Gc_Read_In_I(* TDC *),
				Gc_LuC_Out:= PS[3].Gc.Out.LuC (* Gc_LuC_Out *));
L3_Gc_Read_In_Q:=PSModbus_Out_3.TDC_Read_Out;
L3_Gc_Read_Rsp_Q:=PSModbus_Out_3.TDC_ReadData_Out;
								
(*Line 3 BMS Modbus Out	*)
BMSModbus_Out_3(
					TDC_cmd_I				:=		L3_BMS_Read_In_I ,
					BMS_Sys					:=		PS[3].BMS.Out.LuC.BatSimBMS_Sys,
					TotalRackNbPa			:=		PS[3].BMS.In.Param.TotalRackCntPa,
					BatSim_Rack_Array		:=		PS[3].BMS.Out.LuC.BatSim_Rack_Array
					)	;	
L3_BMS_Read_In_Q			:=	BMSModbus_Out_3.TDC_cmd_Q		;	
L3_BMS_Read_Resp_Q			:=	BMSModbus_Out_3.TDC_mon_Q		;	
BMS3_MB 					:=	BMSModbus_Out_3.BMS_MD		;	
(*_______________________________________________*)
(* Line 4 GC Modbus Out*)
								
PSModbus_Out_4(	TDC_Read_In:=L4_Gc_Read_In_I(* TDC *),
				Gc_LuC_Out:= PS[4].Gc.Out.LuC (* Gc_LuC_Out *));
L4_Gc_Read_In_Q:=PSModbus_Out_4.TDC_Read_Out;
L4_Gc_Read_Rsp_Q:=PSModbus_Out_4.TDC_ReadData_Out;
								
(*Line 4 BMS Modbus Out	*)
BMSModbus_Out_4(
					TDC_cmd_I				:=		L4_BMS_Read_In_I ,
					BMS_Sys					:=		PS[4].BMS.Out.LuC.BatSimBMS_Sys,
					TotalRackNbPa			:=		PS[4].BMS.In.Param.TotalRackCntPa,
					BatSim_Rack_Array		:=		PS[4].BMS.Out.LuC.BatSim_Rack_Array
					)	;	
L4_BMS_Read_In_Q			:=	BMSModbus_Out_4.TDC_cmd_Q		;	
L4_BMS_Read_Resp_Q			:=	BMSModbus_Out_4.TDC_mon_Q		;	
BMS4_MB 					:=	BMSModbus_Out_4.BMS_MD		;					
(*_______________________________________________*)
(* Line 5 GC Modbus Out*)
								
PSModbus_Out_5(	TDC_Read_In:=L5_Gc_Read_In_I(* TDC *),
				Gc_LuC_Out:= PS[5].Gc.Out.LuC (* Gc_LuC_Out *));
L5_Gc_Read_In_Q:=PSModbus_Out_5.TDC_Read_Out;
L5_Gc_Read_Rsp_Q:=PSModbus_Out_5.TDC_ReadData_Out;
								
(*Line 5 BMS Modbus Out	*)
BMSModbus_Out_5(
					TDC_cmd_I				:=		L5_BMS_Read_In_I ,
					BMS_Sys					:=		PS[5].BMS.Out.LuC.BatSimBMS_Sys,
					TotalRackNbPa			:=		PS[5].BMS.In.Param.TotalRackCntPa,
					BatSim_Rack_Array		:=		PS[5].BMS.Out.LuC.BatSim_Rack_Array
					)	;	
L5_BMS_Read_In_Q			:=	BMSModbus_Out_5.TDC_cmd_Q		;	
L5_BMS_Read_Resp_Q			:=	BMSModbus_Out_5.TDC_mon_Q		;	
BMS5_MB 					:=	BMSModbus_Out_5.BMS_MD		;
								
(*_______________________________________________*)
FedMod_Out_1(	Feeder_Out	:=	  Fed_Data[1].Feeder_Out	)	;
Fed_01_PAct_Q	:=	FedMod_Out_1.Fed_01_PAct_Q	;	
Fed_01_EAct_Q	:=	FedMod_Out_1.Fed_01_EAct_Q	;	
Fed_01_EExportAct_Q	:=	FedMod_Out_1.Fed_01_EExportAct_Q	;	
Fed_01_EImportAct_Q	:=	FedMod_Out_1.Fed_01_EImportAct_Q	;	
Fed_01_ExportKvarhAct_Q	:=	FedMod_Out_1.Fed_01_ExportKvarhAct_Q	;	
Fed_01_FAct_Q	:=	FedMod_Out_1.Fed_01_FAct_Q	;	
Fed_01_I1Act_Q	:=	FedMod_Out_1.Fed_01_I1Act_Q	;	
Fed_01_I2Act_Q	:=	FedMod_Out_1.Fed_01_I2Act_Q	;	
Fed_01_I3Act_Q	:=	FedMod_Out_1.Fed_01_I3Act_Q	;	
Fed_01_IAvgAct_Q	:=	FedMod_Out_1.Fed_01_IAvgAct_Q	;	
Fed_01_KvarhAct_Q	:=	FedMod_Out_1.Fed_01_KvarhAct_Q	;	
Fed_01_ImportKvarhAct_Q	:=	FedMod_Out_1.Fed_01_ImportKvarhAct_Q	;	
Fed_01_Line_Q	:=	FedMod_Out_1.Fed_01_Line_Q	;	
Fed_01_PfAct_Q	:=	FedMod_Out_1.Fed_01_PfAct_Q	;	
Fed_01_QAct_Q	:=	FedMod_Out_1.Fed_01_QAct_Q	;	
Fed_01_SAct_Q	:=	FedMod_Out_1.Fed_01_SAct_Q	;	
Fed_01_U123AvgAct_Q	:=	FedMod_Out_1.Fed_01_U123AvgAct_Q	;	
Fed_01_U12Act_Q	:=	FedMod_Out_1.Fed_01_U12Act_Q	;	
Fed_01_U1nAct_Q	:=	FedMod_Out_1.Fed_01_U1nAct_Q	;	
Fed_01_U23Act_Q	:=	FedMod_Out_1.Fed_01_U23Act_Q	;	
Fed_01_U2nAct_Q	:=	FedMod_Out_1.Fed_01_U2nAct_Q	;	
Fed_01_U31Act_Q	:=	FedMod_Out_1.Fed_01_U31Act_Q	;	
Fed_01_U3nAct_Q	:=	FedMod_Out_1.Fed_01_U3nAct_Q	;	
Fed_01_UAct_Q	:=	FedMod_Out_1.Fed_01_UAct_Q	;
							
						
					
END_PROGRAM

CONFIGURATION emC_PPC
  RESOURCE emC_PPC_FUN ON PLC
    VAR_GLOBAL  (* PLCMODE_ON *)
      PLCMODE_ON AT %MX 1.0.0 : BOOL;
      PLCMODE_RUN AT %MX 1.0.1 : BOOL;
      PLCMODE_STOP AT %MX 1.0.2 : BOOL;
      PLCMODE_HALT AT %MX 1.0.3 : BOOL;
      PLCDEBUG_BPSET AT %MX 1.1.4 : BOOL;
      PLCDEBUG_FORCE AT %MX 1.2.0 : BOOL;
      PLCDEBUG_POWERFLOW AT %MX 1.2.3 : BOOL;
      PLC_TICKS_PER_SEC AT %MW 1.44 : INT;
      PLC_SYS_TICK_CNT AT %MD 1.52 : DINT;
      emC_LUC : emC_LUC_Array;
      LUC_Num : INT := 1;
      MbCommTOutPa_S : TIME;
      MessageTimeDelayPa_S : TIME;
      NbOfRackPa_S : INT;
      NbOfBankPa : INT;
      NbOfBankPa_S : INT;
      MapOfRackStruct_S : INT;
      InvDcBusUMinPa : REAL;
      InvDcBusUMinPa_S : REAL;
      BattSysSyncUBiasPa_S : REAL;
      InvDcBusUMaxPa_S : REAL;
      BattRackNomPActPa_S : REAL;
      RacksStartingTimeoutPa_S : TIME;
      Batt_SYSSyncRangePa_S : REAL;
      DrtChrgOnSocLookUpSocPa_S : DerateLookUpPa;
      DrtChrgOnSocLookUpDrtPa_S : DerateLookUpPa;
      DrtDChrgOnSocLookUpSocPa_S : DerateLookUpPa;
      DrtDChrgOnSocLookUpDrtPa_S : DerateLookUpPa;
      DerateTempLookUpTempPa_S : DerateLookUpPa;
      DerateTempLookUpDeratePa_S : DerateLookUpPa;
      RacksStoppingTimeoutPa_S : TIME;
      EnDerateWrtSocPa_S : BOOL;
      EnDerateWrtTempPa_S : BOOL;
      ClockSyncIntervalPa_S : TIME;
      WatchDogModePa_S : INT;
      ClockSyncEnPA_S : BOOL;
      InvPActMaxPa_S : REAL;
      MinPctOfRkPa_S : REAL;
      InvPActMinPa_S : REAL;
      BattRackNomEActPa_S : REAL;
      MapOfRackPa_S : MapOfRackStruct;
      emC_PPC : emC_PPC_Array;
      NbOfLuCPa : INT;
      PPCNum : INT := 1;
      Execute_Cmd : BOOL;
      TestPset : REAL;
      Sys_Data : Sys_Data;
      Sys_Parameters : Sys_Parameters;
      Grid_Dat : Grid_Dat;
      TStep : TIME;
      Synch_Parameters : Synch_Parameters;
      Fed_Data : Feeder_Data;
      PS : Ps_LineUP;
      HMIFeeder_Var_IN : Feeder_Var_IN;
      LuCNum : INT;
    END_VAR
    TASK ?(INTERVAL := 00:00:00.100, PRIORITY := 0);
  END_RESOURCE
END_CONFIGURATION

CONFIGURATION emC_LUC_1
  RESOURCE emC_LUC_FUN ON PLC
    VAR_GLOBAL  (* PLCMODE_ON *)
      PLCMODE_ON AT %MX 1.0.0 : BOOL;
      PLCMODE_RUN AT %MX 1.0.1 : BOOL;
      PLCMODE_STOP AT %MX 1.0.2 : BOOL;
      PLCMODE_HALT AT %MX 1.0.3 : BOOL;
      PLCDEBUG_BPSET AT %MX 1.1.4 : BOOL;
      PLCDEBUG_FORCE AT %MX 1.2.0 : BOOL;
      PLCDEBUG_POWERFLOW AT %MX 1.2.3 : BOOL;
      PLC_TICKS_PER_SEC AT %MW 1.44 : INT;
      PLC_SYS_TICK_CNT AT %MD 1.52 : DINT;
      emC_LUC : emC_LUC_Array;
      LUC_Num : INT;
      MbCommTOutPa_S : TIME;
      MessageTimeDelayPa_S : TIME;
      NbOfRackPa_S : INT;
      NbOfBankPa : INT;
      NbOfBankPa_S : INT;
      MapOfRackStruct_S : INT;
      InvDcBusUMinPa : REAL;
      InvDcBusUMinPa_S : REAL;
      BattSysSyncUBiasPa_S : REAL;
      InvDcBusUMaxPa_S : REAL;
      BattRackNomPActPa_S : REAL;
      RacksStartingTimeoutPa_S : TIME;
      Batt_SYSSyncRangePa_S : REAL;
      DrtChrgOnSocLookUpSocPa_S : DerateLookUpPa;
      DrtChrgOnSocLookUpDrtPa_S : DerateLookUpPa;
      DrtDChrgOnSocLookUpSocPa_S : DerateLookUpPa;
      DrtDChrgOnSocLookUpDrtPa_S : DerateLookUpPa;
      DerateTempLookUpTempPa_S : DerateLookUpPa;
      DerateTempLookUpDeratePa_S : DerateLookUpPa;
      RacksStoppingTimeoutPa_S : TIME;
      EnDerateWrtSocPa_S : BOOL;
      EnDerateWrtTempPa_S : BOOL;
      ClockSyncIntervalPa_S : TIME;
      WatchDogModePa_S : INT;
      ClockSyncEnPA_S : BOOL;
      InvPActMaxPa_S : REAL;
      MinPctOfRkPa_S : REAL;
      InvPActMinPa_S : REAL;
      BattRackNomEActPa_S : REAL;
      MapOfRackPa_S : MapOfRackStruct;
    END_VAR
    TASK ?(INTERVAL := 00:00:00.100, PRIORITY := 0);
  END_RESOURCE
END_CONFIGURATION

CONFIGURATION emC_LUC_2
  RESOURCE emC_LUC_FUN ON PLC
    VAR_GLOBAL  (* PLCMODE_ON *)
      PLCMODE_ON AT %MX 1.0.0 : BOOL;
      PLCMODE_RUN AT %MX 1.0.1 : BOOL;
      PLCMODE_STOP AT %MX 1.0.2 : BOOL;
      PLCMODE_HALT AT %MX 1.0.3 : BOOL;
      PLCDEBUG_BPSET AT %MX 1.1.4 : BOOL;
      PLCDEBUG_FORCE AT %MX 1.2.0 : BOOL;
      PLCDEBUG_POWERFLOW AT %MX 1.2.3 : BOOL;
      PLC_TICKS_PER_SEC AT %MW 1.44 : INT;
      PLC_SYS_TICK_CNT AT %MD 1.52 : DINT;
      emC_LUC : emC_LUC_Array;
      LUC_Num : INT;
      MbCommTOutPa_S : TIME;
      MessageTimeDelayPa_S : TIME;
      NbOfRackPa_S : INT;
      NbOfBankPa : INT;
      NbOfBankPa_S : INT;
      MapOfRackStruct_S : INT;
      InvDcBusUMinPa : REAL;
      InvDcBusUMinPa_S : REAL;
      BattSysSyncUBiasPa_S : REAL;
      InvDcBusUMaxPa_S : REAL;
      BattRackNomPActPa_S : REAL;
      RacksStartingTimeoutPa_S : TIME;
      Batt_SYSSyncRangePa_S : REAL;
      DrtChrgOnSocLookUpSocPa_S : DerateLookUpPa;
      DrtChrgOnSocLookUpDrtPa_S : DerateLookUpPa;
      DrtDChrgOnSocLookUpSocPa_S : DerateLookUpPa;
      DrtDChrgOnSocLookUpDrtPa_S : DerateLookUpPa;
      DerateTempLookUpTempPa_S : DerateLookUpPa;
      DerateTempLookUpDeratePa_S : DerateLookUpPa;
      RacksStoppingTimeoutPa_S : TIME;
      EnDerateWrtSocPa_S : BOOL;
      EnDerateWrtTempPa_S : BOOL;
      ClockSyncIntervalPa_S : TIME;
      WatchDogModePa_S : INT;
      ClockSyncEnPA_S : BOOL;
      InvPActMaxPa_S : REAL;
      MinPctOfRkPa_S : REAL;
      InvPActMinPa_S : REAL;
      BattRackNomEActPa_S : REAL;
      MapOfRackPa_S : MapOfRackStruct;
    END_VAR
    TASK ?(INTERVAL := 00:00:00.100, PRIORITY := 0);
  END_RESOURCE
END_CONFIGURATION

CONFIGURATION emC_LUC_3
  RESOURCE emC_LUC_FUN ON PLC
    VAR_GLOBAL  (* PLCMODE_ON *)
      PLCMODE_ON AT %MX 1.0.0 : BOOL;
      PLCMODE_RUN AT %MX 1.0.1 : BOOL;
      PLCMODE_STOP AT %MX 1.0.2 : BOOL;
      PLCMODE_HALT AT %MX 1.0.3 : BOOL;
      PLCDEBUG_BPSET AT %MX 1.1.4 : BOOL;
      PLCDEBUG_FORCE AT %MX 1.2.0 : BOOL;
      PLCDEBUG_POWERFLOW AT %MX 1.2.3 : BOOL;
      PLC_TICKS_PER_SEC AT %MW 1.44 : INT;
      PLC_SYS_TICK_CNT AT %MD 1.52 : DINT;
      emC_LUC : emC_LUC_Array;
      LUC_Num : INT;
      MbCommTOutPa_S : TIME;
      MessageTimeDelayPa_S : TIME;
      NbOfRackPa_S : INT;
      NbOfBankPa : INT;
      NbOfBankPa_S : INT;
      MapOfRackStruct_S : INT;
      InvDcBusUMinPa : REAL;
      InvDcBusUMinPa_S : REAL;
      BattSysSyncUBiasPa_S : REAL;
      InvDcBusUMaxPa_S : REAL;
      BattRackNomPActPa_S : REAL;
      RacksStartingTimeoutPa_S : TIME;
      Batt_SYSSyncRangePa_S : REAL;
      DrtChrgOnSocLookUpSocPa_S : DerateLookUpPa;
      DrtChrgOnSocLookUpDrtPa_S : DerateLookUpPa;
      DrtDChrgOnSocLookUpSocPa_S : DerateLookUpPa;
      DrtDChrgOnSocLookUpDrtPa_S : DerateLookUpPa;
      DerateTempLookUpTempPa_S : DerateLookUpPa;
      DerateTempLookUpDeratePa_S : DerateLookUpPa;
      RacksStoppingTimeoutPa_S : TIME;
      EnDerateWrtSocPa_S : BOOL;
      EnDerateWrtTempPa_S : BOOL;
      ClockSyncIntervalPa_S : TIME;
      WatchDogModePa_S : INT;
      ClockSyncEnPA_S : BOOL;
      InvPActMaxPa_S : REAL;
      MinPctOfRkPa_S : REAL;
      InvPActMinPa_S : REAL;
      BattRackNomEActPa_S : REAL;
      MapOfRackPa_S : MapOfRackStruct;
    END_VAR
    TASK ?(INTERVAL := 00:00:00.100, PRIORITY := 0);
  END_RESOURCE
END_CONFIGURATION

CONFIGURATION emC_LUC_4
  RESOURCE emC_LUC_FUN ON PLC
    VAR_GLOBAL  (* PLCMODE_ON *)
      PLCMODE_ON AT %MX 1.0.0 : BOOL;
      PLCMODE_RUN AT %MX 1.0.1 : BOOL;
      PLCMODE_STOP AT %MX 1.0.2 : BOOL;
      PLCMODE_HALT AT %MX 1.0.3 : BOOL;
      PLCDEBUG_BPSET AT %MX 1.1.4 : BOOL;
      PLCDEBUG_FORCE AT %MX 1.2.0 : BOOL;
      PLCDEBUG_POWERFLOW AT %MX 1.2.3 : BOOL;
      PLC_TICKS_PER_SEC AT %MW 1.44 : INT;
      PLC_SYS_TICK_CNT AT %MD 1.52 : DINT;
      emC_LUC : emC_LUC_Array;
      LUC_Num : INT;
      MbCommTOutPa_S : TIME;
      MessageTimeDelayPa_S : TIME;
      NbOfRackPa_S : INT;
      NbOfBankPa : INT;
      NbOfBankPa_S : INT;
      MapOfRackStruct_S : INT;
      InvDcBusUMinPa : REAL;
      InvDcBusUMinPa_S : REAL;
      BattSysSyncUBiasPa_S : REAL;
      InvDcBusUMaxPa_S : REAL;
      BattRackNomPActPa_S : REAL;
      RacksStartingTimeoutPa_S : TIME;
      Batt_SYSSyncRangePa_S : REAL;
      DrtChrgOnSocLookUpSocPa_S : DerateLookUpPa;
      DrtChrgOnSocLookUpDrtPa_S : DerateLookUpPa;
      DrtDChrgOnSocLookUpSocPa_S : DerateLookUpPa;
      DrtDChrgOnSocLookUpDrtPa_S : DerateLookUpPa;
      DerateTempLookUpTempPa_S : DerateLookUpPa;
      DerateTempLookUpDeratePa_S : DerateLookUpPa;
      RacksStoppingTimeoutPa_S : TIME;
      EnDerateWrtSocPa_S : BOOL;
      EnDerateWrtTempPa_S : BOOL;
      ClockSyncIntervalPa_S : TIME;
      WatchDogModePa_S : INT;
      ClockSyncEnPA_S : BOOL;
      InvPActMaxPa_S : REAL;
      MinPctOfRkPa_S : REAL;
      InvPActMinPa_S : REAL;
      BattRackNomEActPa_S : REAL;
      MapOfRackPa_S : MapOfRackStruct;
    END_VAR
    TASK ?(INTERVAL := 00:00:00.100, PRIORITY := 0);
  END_RESOURCE
END_CONFIGURATION

CONFIGURATION emC_LUC_5
  RESOURCE emC_LUC_FUN ON PLC
    VAR_GLOBAL  (* PLCMODE_ON *)
      PLCMODE_ON AT %MX 1.0.0 : BOOL;
      PLCMODE_RUN AT %MX 1.0.1 : BOOL;
      PLCMODE_STOP AT %MX 1.0.2 : BOOL;
      PLCMODE_HALT AT %MX 1.0.3 : BOOL;
      PLCDEBUG_BPSET AT %MX 1.1.4 : BOOL;
      PLCDEBUG_FORCE AT %MX 1.2.0 : BOOL;
      PLCDEBUG_POWERFLOW AT %MX 1.2.3 : BOOL;
      PLC_TICKS_PER_SEC AT %MW 1.44 : INT;
      PLC_SYS_TICK_CNT AT %MD 1.52 : DINT;
      emC_LUC : emC_LUC_Array;
      LUC_Num : INT;
      MbCommTOutPa_S : TIME;
      MessageTimeDelayPa_S : TIME;
      NbOfRackPa_S : INT;
      NbOfBankPa : INT;
      NbOfBankPa_S : INT;
      MapOfRackStruct_S : INT;
      InvDcBusUMinPa : REAL;
      InvDcBusUMinPa_S : REAL;
      BattSysSyncUBiasPa_S : REAL;
      InvDcBusUMaxPa_S : REAL;
      BattRackNomPActPa_S : REAL;
      RacksStartingTimeoutPa_S : TIME;
      Batt_SYSSyncRangePa_S : REAL;
      DrtChrgOnSocLookUpSocPa_S : DerateLookUpPa;
      DrtChrgOnSocLookUpDrtPa_S : DerateLookUpPa;
      DrtDChrgOnSocLookUpSocPa_S : DerateLookUpPa;
      DrtDChrgOnSocLookUpDrtPa_S : DerateLookUpPa;
      DerateTempLookUpTempPa_S : DerateLookUpPa;
      DerateTempLookUpDeratePa_S : DerateLookUpPa;
      RacksStoppingTimeoutPa_S : TIME;
      EnDerateWrtSocPa_S : BOOL;
      EnDerateWrtTempPa_S : BOOL;
      ClockSyncIntervalPa_S : TIME;
      WatchDogModePa_S : INT;
      ClockSyncEnPA_S : BOOL;
      InvPActMaxPa_S : REAL;
      MinPctOfRkPa_S : REAL;
      InvPActMinPa_S : REAL;
      BattRackNomEActPa_S : REAL;
      MapOfRackPa_S : MapOfRackStruct;
    END_VAR
    TASK ?(INTERVAL := 00:00:00.100, PRIORITY := 0);
  END_RESOURCE
END_CONFIGURATION

CONFIGURATION emC_Sim
  RESOURCE emC_Sim_FUN ON PLC
    VAR_GLOBAL  (* PS *)
      PS : Ps_LineUP;
      PLCMODE_ON AT %MX 1.0.0 : BOOL;
      PLCMODE_RUN AT %MX 1.0.1 : BOOL;
      PLCMODE_STOP AT %MX 1.0.2 : BOOL;
      PLCMODE_HALT AT %MX 1.0.3 : BOOL;
      PLCDEBUG_BPSET AT %MX 1.1.4 : BOOL;
      PLCDEBUG_FORCE AT %MX 1.2.0 : BOOL;
      PLCDEBUG_POWERFLOW AT %MX 1.2.3 : BOOL;
      PLC_TICKS_PER_SEC AT %MW 1.44 : INT;
      PLC_SYS_TICK_CNT AT %MD 1.52 : DINT;
      Sys_Data : Sys_Data;
      HMIFeeder_Var_IN : Feeder_Var_IN;
      Sys_Parameters : Sys_Parameters;
      Grid_Dat : Grid_Dat;
      Synch_Parameters : Synch_Parameters;
      TStep : TIME;
      Fed_Data : Feeder_Data;
      emC_LUC : emC_LUC_Array;
      LuNumPa : INT;
    END_VAR
    TASK ?(INTERVAL := 00:00:00.100, PRIORITY := 0);
  END_RESOURCE
END_CONFIGURATION
